		// INV Measures from Datalogger
		MesP 				: REAL ; 		(* (kW) 	Active Power output (AC) of inverter PCS01*)
		MesQ 				: REAL ;  		(* (kVAr)   Reactive AC Power Produced				  *)
		MesPdc 				: REAL ;  		(* (kW) 	Power measure (DC) of inverter			  *)
		MesIdc 				: REAL ;	 	(* (A) 	    Total Current measure (DC)				  *)
		MesUdc 				: REAL ;  		(* (V)  	Mean Voltage measure (DC)				  *)
		MesU 				: REAL ;		(* (V) 	    Mean Voltage measure (AC)				  *)
		MesV				: REAL ; 		(* (V)      Mean Phase to Neutral voltage			  *)
		MesI				: REAL ;		(* (A)      Mean Phase Current						  *)
		MesI0               : REAL ;        (* (A) 		Residual current						  *) 
		MesFreq				: REAL ; 		(* (Hz)     Frequency                                 *)
		MesS				: REAL ; 		(* (kVA)     Apparent Power						      *)
		MesInsuResistor		: REAL ; 		(* (kOhms) Insulation Resistance					  *)
		MesCosPhi			: REAL ; 		(* (p.u) Power Factor								  *)
		MesTemp				: REAL ; 		(* (C) Inverter Temperature							  *)
		MesState_Inv		: UINT ;		(* (NA) Inverter Status								  *)
		ParamPn				: REAL ; 		(* (kW) Nominal Capacity of SMA 25000 TL Inverter	  *)
		ParamQn				: REAL ;		(* (kVAr) Nominal reactive power 					  *)
		MesCurtl		    : BOOL ; 		(* (NA)Cal True if the inverter is curtailing Power	  *)
		MesAlarmCom			: BOOL ; 		(* (NA) Communication Alarm							  *)
		MesCP_Read			: BOOL := TRUE;	(* (NA) Cal : Permanent Condition for Read			  *)
		MesCP_Write			: BOOL := FALSE;	(* (NA) Cal : Permanenent Condition for Write		  *)
		                                                                                        
		MesOpened_Ac        : BOOL ;   		(* (NA) Ac switch is opened							  *)
		MesOpened_Dc        : BOOL ;   		(* (NA) Dc switch is opened							  *)
		                                                                                        
		OUT_CmdStart        : BOOL ;        (* (NA) OUT start command 							  *)
		OUT_CmdStop         : BOOL ;        (* (NA) OUT stop command   							  *)
		OUT_SetptPLimit    	: REAL ;        (* (kW) OUT P setpoint  							  *)
		OUT_SetptQ          : REAL ;        (* (kVAr)  OUT Q setpoint   						  *)
		MesState			: WORD ; 		(* (NA) Cal: Akuo Internal State . O=Stopped, 1 = RUN, 2 = Curtailment *)
		MesAlarmCode		: WORD ; 		(* (NA) Internal Akuo AlarmCode                       *)
		MesWarningCode		: WORD ; 		(* (NA) Internal Akuo WarningCode                     *)
		MesEventCode		: WORD ; 		(* (NA) Internal Akuo EventCode                       *)

END_STRUCT
END_TYPE

// ---- 01_Equipement_Library/Inverter/INV_DcModule.TcDUT
TYPE INV_DcModule :
STRUCT
	MesIdc				: REAL ; (* (A) Current of the Dc Module *)
	MesUdc				: REAL ; (* (V) Voltage of the Dc Module *)
	MesPdc				: REAL ; (* (kW) Power of the Dc Module *)
	MesClosed_DcSwitch	: BOOL ; (* (NA) Status of DC switch*)
	MesChargedSpring	: BOOL ; (* (NA) Status of string of DC switch*)
         		
	AX_STR				: ARRAY[1..CstNbSB_DcModule_G] OF STR;
END_STRUCT
END_TYPE

// ---- 01_Equipement_Library/Inverter/INV_DU.TcDUT
///////////
// Structure For Module. Main Operating Data to be saved (ex: OPC).  
//////////
TYPE INV_DU :
STRUCT
	
		MesI 				: REAL ; 		(* (dA) DU Current *)
		MesU 				: REAL ;  		(* (dV) DU Voltage *)
		MesIDState			: UINT ;		(* (NA) DU Status  *)
		
END_STRUCT
END_TYPE

// ---- 01_Equipement_Library/Inverter/INV_ABB_PVS.TcDUT
TYPE INV_ABB_PVS :
STRUCT
	MesData				: INV;		(* INV Object 									*)
	
	AX_STR				: ARRAY[1..12] OF STR;	(* STR Object 						*)
	
	MesI1				: REAL;		(* (A) Current Phase 1 							*)
	MesI2				: REAL;     (* (A) Current Phase 2 							*)
	MesI3				: REAL;     (* (A) Current Phase 3 							*)
	MesV1				: REAL;     (* (V) Voltage Phase 1 							*)
	MesV2				: REAL;     (* (V) Voltage Phase 2 							*)
	MesV3				: REAL;     (* (V) Voltage Phase 3 							*)
	MesU12				: REAL;     (* (V) Voltage between Phase 1 and 2 			*)
	MesU23				: REAL;     (* (V) Voltage between Phase 2 and 3 			*)
	MesU31				: REAL;     (* (V) Voltage between Phase 1 and 3 			*)
	MesPF				: REAL;     (* (NA) Power Factor							*)
	                                                                        		
	MesTemp_AC_cab		: REAL;		(* (C) Cabinet Temperature						*)
	MesTemp_HeatSink	: REAL;		(* (C) Heat Sink Temperature					*)
	MesState_InvWord	: WORD;		(* (NA)											*)
	MesVndOpeState		: UINT;		(* (NA) 										*)
	MesGlobalEvt		: WORD;		(* (NA) 										*)
	MesEacTot			: ULINT;	(* (NA) 										*)	
	MesEacDay			: LREAL;    (* (NA) 										*)
	
	MesEvent1 			: WORD;		(* (NA)											*)
	MesEventBitFld2 	: WORD;		(* (NA)											*)
	MesVndEventBitFld1 	: WORD;		(* (NA)											*)
	MesVndEventBitFld2 	: WORD;		(* (NA)											*)
	MesVndEventBitFld3 	: WORD;		(* (NA)											*)
	
	
	CmdP_Ack			: BOOL := TRUE;	(* (NA) P Command Acknowledge 				*)
	CmdQ_Ack			: BOOL := TRUE;	(* (NA) Q Command Acknowledge 				*)
	CmdPF_Ack			: BOOL;			(* (NA) Power Factor Command Acknowledge 	*)
	CmdStart_Ack		: BOOL := TRUE;	(* (NA) Start Command Acknowledge 			*)
	OUT_SetptCosPhi		: REAL := 1;	(* (NA) Power factor SetPoint Acknowledge	*)
	
END_STRUCT
END_TYPE

// ---- 01_Equipement_Library/Inverter/INV_Huawei.TcDUT
///////////
// Structure For Inverter. Main Operating Data to be saved ( ex: OPC ) .  
//////////
TYPE INV_Huawei :
STRUCT
	
	// INV Measures
		MesData				: INV ; (* INV *) 
                        	
		STR					: ARRAY[1..CstNbSB_INV_G ] OF STR ;  	(* STR *) 
		                	
		MesEDay				: REAL ;	    			(* (kWh)Daily Energy	*)
	    MesETot				: REAL ;					(* (kWh)Total Energy	*)
		MesI1				: REAL ;					(*	(A) MesI1			*)
		MesI2				: REAL ;					(*	(A) MesI2			*)
	    MesI3				: REAL ;					(*	(A) MesI3			*)
		MesU12				: REAL ;					(*	(V) MesU12			*)
        MesU23				: REAL ;					(*	(V) MesU23			*)
        MesU31				: REAL ;					(*	(V) MesU31			*)
		MesV1				: REAL ;					(*	(V) MesV1			*)
		MesV2				: REAL ;					(*	(V) MesV2			*)
		MesV3				: REAL ;					(*	(V) MesV3			*)
                        	                			
		MesStateIndic		: WORD ;					(*	(NA) Device status 		*)
		MesDeviceStatus		: WORD ;
// 0: standby , 1:grid connected , 2: grid connected normally , 3 : grid connection with derating due to power rationing , 4 grid connection with derating due to internal causes of the solar inverter
// 5 : normal stop , 6 : stop due to fault , 7 : stop due to power rationning , 8 : shutdown , 9 : spot check 


		MesOpeStatus 		: WORD ;					(*	(NA) MesOpeStatus 		*)
// 0 : locking status (0: locked; 1: unlocked) - 1 : PV Connection sttaus , 2 : DSP Data collection , 

		MesAlm1				: WORD ;					(*	(NA) MesAlm1				*)
		MesAlm2				: WORD ;					(*	(NA) MesAlm2				*)
		MesAlm3				: WORD ;					(*	(NA) MesAlm3				*)
	                                                        	
		MesID_DevStatus1	: WORD;						(* (NA) Akuo Created satus to compute device status alarms*)
		MesID_DevStatus2	: WORD;						(* (NA) Akuo Created satus to compute device status alarms*)
		


END_STRUCT
END_TYPE

// ---- 01_Equipement_Library/Inverter/INV_PE_HEMK.TcDUT
   ///////////
// Structure for PE Inverter. Main Operating Data to be saved (ex: OPC).  
//////////
TYPE INV_PE_HEMK:
STRUCT
	
	MesData					: INV ;				(* (NA) MesData*) 		            		
	// INV Measures
	AX_PowerCol				: ARRAY[1..CstNbPowerCol_INV_G ] OF PowerCol_INV_PE_HEMK; 			(* (NA) INV power columns *)
	AX_DcModule				: ARRAY[1..CstNbDcModule_INV_G] OF INV_DcModule; 			(* (NA) DC Inputs to the Inverter*)	
	
		
	//Electrical Measurements	
	MesAcDay				: UINT;				(* (kWh) Daily energy*)
	MesAcTot				: UINT;				(* (kWh) Total energy*)

	
	MesI1					: REAL; 			(* (A) Current phase 1 (R). INV: SV1.4 Grid current I1 (HEMK)															*)
	MesI2					: REAL; 			(* (A) Current phase 2 (S). INV: SV1.5 Grid current I2 (HEMK)															*)
	MesI3					: REAL; 			(* (A) Current phase 3 (T). INV: SV1.6 Grid current I3  (HEMK)															*)
	MesU12					: REAL; 			(* (V) Phase AB RMS voltage (line to line)at grid side of AC circuit breaker CB501. INV: SV1.1 Grid voltage RS (HEMK)	*)
	MesU23					: REAL; 			(* (V) Phase BC RMS voltage (line to line)at grid side of AC circuit breaker CB501. INV: SV1.2 Grid voltage ST(HEMK)	*)
	MesU31					: REAL; 			(* (V) Phase CA RMS voltage (line to line)at grid side of AC circuit breaker CB501. INV: SV1.3 Grid voltage TR (HEMK)	*)
	MesStatusCurtail_P		: WORD; 			(* (NA) P control : Cause of P control*)
	MesStatusCurtail_Q		: WORD; 			(* (NA) Q control : Cause of Q control*)
	MesDeratingGlobal		: REAL;				(* (%) Derating global taking into consideration IGBT Temp, Vdc et admission temp*)                               			
	                                			
	//Status Summary                			
	MesEventID				: REAL;				(* (NA) Event ID of the currently active event. 0= No event, 1 = Emergency stop, 3 = Remote emergency stop. SV8.15      *)
	MesIDFault				: UINT;				(* (NA) current fault ID check complete list in tab Failures*)	
	MesIDLastFaultedPowerCol: UINT;				(* (NA) Power Column ID of last alarm communicated*)	
	MesIDWarning			: UINT;				(* (NA) ID of current Warning : check complete list in tab Warnings*)	
	MesStateStart_Freq		: BOOL;				(* (NA) Start conditions Freq : True = Start OK*)
	MesStateStart_Vdc		: BOOL;				(* (NA) Start conditions Vdc : True = Start OK*)
	MesStateStart_MVCells	: BOOL;				(* (NA) Start conditions MVCells : True = Start OK*)
	MesStateStart_P			: BOOL;				(* (NA) Start conditions P : True = Start OK*)
	MesStateStart_Bbox		: BOOL;				(* (NA) Start conditions Bbox : True = Start OK*)
	
                            			
	MesSetptP				: REAL;				(* (%) Measurement of active power setpoint. INV: G8.1.3 P reference  	                                                *)                        	 
	MesSetptQ				: REAL;				(* (%) Measurement of reactive power setpoint. INV: G8.1.4 Q reference	                                   	            *)
	
	// System Commands
	ParamID_QMode			: UINT := 1; 		(* (NA) reactive power control mode : 0: Cos Phi, 1: Q,  2: I, 4: V/Q mode   G8.1.2 register: 40551  		*)
	ParamID_PMode			: UINT := 1; 		(* (NA) active power control mode : 0: MPPt, 1: I, 2: P, 3: Vdc										 		*)
		                                    	                                                                                                         		
	MesCP_Start        		: BOOL;				(* (NA) Start conditions. INV: SV4.3.1-Start conditions all											 		*)                 		        		
	                                                                                                         											
	// Inverter's Control Cabinet  Status                                                                       											
	MesTemp_Internal		: REAL; 		 	(* (C) Control cabinet temperature. INV: SV4.1.4 Internal temperature										*)
	MesTemp_Control			: REAL; 		 	(* (C) Control cabinet temperature. INV: SV4.1.4 Internal temperature										*)
	MesTemp_IGBTmax			: REAL; 		 	(* (C) Maximum IGBT temperature. INV: SV4.1.5 Max IGBTs temperature											*)
	MesTemp_PowerColmax		: REAL; 		 	(* (C) Maximum power column temperature. INV: SV4.1.6 Max modules temperature								*)
	MesAlarm_Control		: UINT;			 	(* (NA) Control cabinet alarm. INV: SV4.1.1 Current fault 													*) 
	MesWarning_Control		: UINT;			 	(* (NA) Control cabinet warning. INV: SV4.1.2 Current warning					    						*)			
	MesState_Control 		: UINT;			 	(* (NA) Control cabinet state. INV: SV4.1.3 Current status													*)
	MesState_Module			: WORD;				(* (NA) Status of modules*)	 
	MesNbRunningModules		: UINT;				(* (NA) Number of running modules*)
                                        	                                                    	                                						
	// Reset command                         	                                                    	                                						
	OUT_CmdReset 			: BOOL; 		 	(* (NA) OUT reset command. INV: Reset command 43012															*)

	MesP_LV					: REAL;				(* (kW) LV Active Power*)
	MesQ_LV					: REAL;				(* (kVAr) LV Reactive Power*)
	MesS_LV					: REAL;				(* (kVA) LV Apparent Power*)
	MesCosPhi_LV			: REAL;				(* (NA) LV CosPhi*)
    MesU12_LV				: REAL; 			(* (kV) LV Voltage 12*)                                                                              															
    MesU23_LV				: REAL; 			(* (kV) LV Voltage 23*)                                                                              															
    MesU31_LV				: REAL; 			(* (kV) LV Voltage 31*)                                                                              															
	MesI1_LV				: REAL; 			(* (A) Current phase 1 (R). INV: SV1.4 Grid current I1 (HEMK)															*)
	MesI2_LV				: REAL; 			(* (A) Current phase 2 (S). INV: SV1.5 Grid current I2 (HEMK)															*)
	MesI3_LV				: REAL; 			(* (A) Current phase 3 (T). INV: SV1.6 Grid current I3  (HEMK)															*)
	MesPAvailable			: REAL;
	MesPn					: REAL;

	
	MesEventCode2			: WORD ; 


END_STRUCT
END_TYPE

// ---- 01_Equipement_Library/Inverter/INV_PE_HEMG3.TcDUT
///////////
// Structure for PE Inverter. Main Operating Data to be saved (ex: OPC).  
//////////
TYPE INV_PE_HEMG3:
STRUCT
	
	// INV Measures
	MesData					: INV ;	(* (NA) MesData 																										*) 		            		
	// Power column (PE name : Modules) 
	AX_PowerCol				: ARRAY[1..6] OF PowerCol_INV_PE_HEMG3;	(* (NA) Power column of the PE Skid  *) 
	AX_DU 					: ARRAY[1..CstNb_DU_G] OF INV_DU; (* (NA) Disconnecting Units Channels *)
	
	//Electrical Measurements	
	MesI1					: REAL; (* (A) Current phase 1 (R). INV: SV1.4 Grid current I1 (HEMK)															*)
	MesI2					: REAL; (* (A) Current phase 2 (S). INV: SV1.5 Grid current I2 (HEMK)															*)
	MesI3					: REAL; (* (A) Current phase 3 (T). INV: SV1.6 Grid current I3  (HEMK)															*)
	MesU12					: REAL; (* (V) Phase AB RMS voltage (line to line)at grid side of AC circuit breaker CB501. INV: SV1.1 Grid voltage RS (HEMK)	*)
	MesU23					: REAL; (* (V) Phase BC RMS voltage (line to line)at grid side of AC circuit breaker CB501. INV: SV1.2 Grid voltage ST(HEMK)	*)
	MesU31					: REAL; (* (V) Phase CA RMS voltage (line to line)at grid side of AC circuit breaker CB501. INV: SV1.3 Grid voltage TR (HEMK)	*)
	MesPconnected			: REAL; (* (%) Current available active power. INV: SV4.2.1 P limit inst 														*)                                                     									
	MesStatusCurtail_P		: WORD; 			(* (NA) P control : Cause of P control*)
	MesStatusCurtail_Q		: WORD; 			(* (NA) Q control : Cause of Q control*)
	MesInsuResistor_AC		: REAL;	(* (Ohms) AC Insulation Resistance. INV: SV3.2.2  Resistor 																*)
	OUT_CmdInvLocal			: BOOL; (*determine whether setpoint is from local or remote *)
	
	
	
	//Communication Status                                                                                              									
	MesStateCom				: BOOL; (* (NA) Cal: False := Not communicating, True := Communicating	 														*)
	
	//Status Summary
	MesStateCBac			: BOOL; (* (NA) False := Open, True := Close, Status of event139 "CB501 Closed". AC circuit breaker CB501 is closed 			*)
	MesStateCBdc			: BOOL; (* (NA) False := Open, True := Close, Status of event140 "CB201 Closed". DC circuit breaker CB201 is closed             *)
	MesEarthing_Relay		: BOOL; (* (NA) False := Open, True := Close, Status of event157 "K202 Closed". Ground relay K202 is closed                     *)
	MesFaultGnd				: BOOL; (* (NA) False := Alert, True := No alert, Ground fault status. Digital outputDO_121 follows the state of this register  *)
	MesStateNoAlert			: BOOL; (* (NA) False := Alert iverter has detected an abnormal event which prevents operation. ; True := No alert.             *)
	MesState				: UINT; (* (NA) This parameter should be used for informational status only                                                     *)
	MesAlarmID				: UINT; (* (NA) Fallo actual *)
	MesWarningID			: UINT; (* (NA) Warning actual*)


	MesBdrigeCtlMod			: UINT;	(* (NA) Inverter bridge control mode                                                                                    *)
	MesWorkingHr			: REAL; (* (Hr) Total duration that the inverter has been online since power up                                                 *)
	MesEventID				: REAL;	(* (NA) Event ID of the currently active event. 0= No event, 1 = Emergency stop, 3 = Remote emergency stop. SV8.15      *)
	
	MesSetptP				: REAL;	(* (%) Measurement of active power setpoint. INV: G8.1.3 P reference  	                                                *)                        	 
	MesSetptQ				: REAL;	(* (%) Measurement of reactive power setpoint. INV: G8.1.4 Q reference	                                   	            *)
	MesSetptCosPhi			: REAL; (* (pu) Measurement of power factor setpoint. INV: G8.1.4 Cos phi reference                                	            *)
	MesStartDisabled		: BOOL; (* (NA) Start disable : False := Start can be abled 						 											*)
	
	// System Commands
	ParamID_QMode			: UINT := 1; 		(* (NA) reactive power control mode : 0: Cos Phi, 1: Q,  2: I, 4: V/Q mode   G8.1.2 register: 40551  		*)
	ParamID_PMode			: UINT := 1; 		(* (NA) active power control mode : 0: MPPt, 1: I, 2: P, 3: Vdc										 		*)
		                                    	                                                                                                         		
	MesCP_Start        		: BOOL;				(* (NA) Start conditions. INV: SV4.3.1-Start conditions all											 		*)                 		        		
	                                                                                                         											
	// Inverter's Control Cabinet  Status                                                                       											
	MesTemp_DU				: REAL;			 	(* (C) Disconnecting unit temperature. INV: SV4.1.4b DU Internal  											*)
	MesTemp_Control			: REAL; 		 	(* (C) Control cabinet temperature. INV: SV4.1.4 Internal temperature										*)
	MesTemp_IGBTmax			: REAL; 		 	(* (C) Maximum IGBT temperature. INV: SV4.1.5 Max IGBTs temperature											*)
	MesTemp_PowerColmax		: REAL; 		 	(* (C) Maximum power column temperature. INV: SV4.1.6 Max modules temperature								*)
	MesAlarm_Control		: UINT;			 	(* (NA) Control cabinet alarm. INV: SV4.1.1 Current fault 													*) 
	MesWarning_Control		: UINT;			 	(* (NA) Control cabinet warning. INV: SV4.1.2 Current warning					    						*)			
	MesState_Control 		: UINT;			 	(* (NA) Control cabinet state. INV: SV4.1.3 Current status													*)
	                                         	                                                    	                                						
	// Reset command                         	                                                    	                                						
	OUT_CmdReset 			: BOOL; 		 	(* (NA) OUT reset command. INV: Reset command 43012															*)
	OUT_CmdEmergencyStop	: BOOL; 		 	(* (NA) OUT emergency stop command. INV: Emergengy stop command 43200										*) 
	MesNbRunningModules		: REAL; 			(* (NA) Number of modules running*)

    MesEventCode2			: WORD ;                                                                                     															
END_STRUCT
END_TYPE

// ---- 01_Equipement_Library/Inverter/SKID_PE_HEMG3.TcDUT
///////////
// Structure for PE SKID. Main Operating Data to be saved (ex: OPC).  
//////////
TYPE SKID_PE_HEMG3:
STRUCT
	
	MesCP_Read							: BOOL := TRUE;		(* (NA) Cal : Permanent Condition for Read		*)
	MesCP_Write							: BOOL := TRUE;		(* (NA) Cal : Permanenent Condition for Write   *)
	
	MesDisparoTemp_Transformador1 		: BOOL; (* (NA) alarm transformer*)
	MesAlarmTemp_Transformador1	 		: BOOL; (* (NA) warning temp transformer*)
	MesDisparoPresion_Transformador1 	: BOOL; (* (NA) alarm pressure transformer*)
	MesDisparoOil_Transformador1 		: BOOL; (* (NA) alarm oil transformer*)

	MesDisparoTemp_Transformador2 		: BOOL; (* (NA) alarm transformer*)
	MesAlarmTemp_Transformador2	 		: BOOL; (* (NA) warning temp transformer*)
	MesDisparoPresion_Transformador2 	: BOOL; (* (NA) alarm pressure transformer*)
	MesDisparoOil_Transformador2 		: BOOL; (* (NA) alarm oil transformer*)

	MesSeccionador1_Abierto				: BOOL; (* (NA) Secc opened*)
	MesEarth1_Abierto					: BOOL; (* (NA) Earth switch Opened opened*)
	MesMonitorGas						: BOOL; (* (NA) *)
	MesMonitorGas2						: BOOL; (* (NA) *)
	MesSeccionador2_Abierto				: BOOL; (* (NA) Secc opened*)
	MesEarth2_Abierto					: BOOL; (* (NA) Earth switch Opened opened*)
	MesSeccionadorMain1_Abierto			: BOOL; (* (NA) Secc opened*)
	MesEarthMain1_Abierto				: BOOL; (* (NA) Earth switch Opened opened*)
	MesCb1_Abierto						: BOOL; (* (NA) Circuit breaker*)
	MesProtectRelay1_fallo				: BOOL; (* (NA) protect relay fault*)
	MesProtectRelay1_overvoltage		: BOOL; (* (NA) protect relay fault*)
	MesProtectRelay1_springloaded		: BOOL; (* (NA) *)

	MesSeccionadorMain2_Abierto			: BOOL; (* (NA) Secc opened*)
	MesEarthMain2_Abierto				: BOOL; (* (NA) Earth switch Opened opened*)
	MesCb2_Abierto						: BOOL; (* (NA) Circuit breaker*)
	MesProtectRelay2_fallo				: BOOL; (* (NA) protect relay fault*)
	MesProtectRelay2_overvoltage		: BOOL; (* (NA) protect relay fault*)
	MesProtectRelay2_springloaded		: BOOL; (* (NA) *)

	MesTemp1							: REAL;(* (°C) temperature of the transformer*)
	MesTemp2							: REAL;(* (°C) temperature of the transformer*)
	
	MesAlarmCom							: BOOL;
	MesAlarmCode						: WORD; 			(* (NA) Internal Akuo AlarmCode                 *)
	MesWarningCode						: WORD; 			(* (NA) Internal Akuo WarningCode               *)
	MesEventCode						: WORD;		 		(* (NA) Internal Akuo EventCode                 *)                                                                            															
END_STRUCT
END_TYPE

// ---- 01_Equipement_Library/Inverter/PowerCol_INV_PE_HEMK.TcDUT
///////////
// Structure For Module. Main Operating Data to be saved (ex: OPC).  
//////////
TYPE PowerCol_INV_PE_HEMK :
STRUCT
		MesData				: PowerCol_INV ; 	
		
		
		MesS 				: REAL ;  		(* (kVA)   Apparent power output of the power column 													*)
		MesU12				: REAL ;		(* (A) 		Module Voltage																				*)
		MesU23				: REAL ;		(* (A) 		Module Voltage																				*)
		MesU31				: REAL ;		(* (A) 		Module Voltage																				*)
		
		ParamUn				: REAL ;		(* (V) 		Nominal AC voltage (SV4.4.4.1.2)																		*)
		ParamImax			: REAL ; 		(* (A) 		Nominal AC current (SV4.4.4.1.7)																		*) 
		ParamVdcn			: REAL ;        (* (V) 		Nominal DC voltage (SV4.4.4.1.6)																		*)
		ParamIdcmax			: REAL ;        (* (A) 		Nominal DC current (SV4.4.4.1.8)																		*)
		ParamSn				: REAL ;        (* (kVA) 	Nominal apparent power (SV4.4.4.1.3)																	*)
		
		MesTemp				: REAL ;		(* (C) 		Ambient temperature of the selected module																*)
		MesTempmax			: REAL ;		(* (C) 		Maximum IGBT temperature of the selected module															*)
		MesHygro			: REAL ; 		(* (%) 		Percentage of humidity																					*)
		
		MesStateIO			: WORD ;		(* (NA) 	0: Open, 1: Closed. Bit 1 =  fan contactor, Bit 2 = main AC contactor, Bit 3 = AC soft charge contactor, Bit 4 = LCL filter contactor, Bit 5 = DC contactor , Bit 6 = reserved, Bit 7 = if open : overheating in the coil, Bit 8 = fan contactor feedback, Bit 9 = AC main contactor feedback, Bit 10 = AC soft charge contactor feedback, Bit 11 = LCL filter contactor feedback , Bit 12 = DC contactor feedback *) 		
		MesState			: UINT ;		(* (NA) 	Module status (SV9.3 PE documentation p.97)																*)
		
		MesEActProd			: REAL ;		(* (kWh) 	Total amount of  generated energy since commissioning 													*)
		MesEReactProd		: REAL ;		(* (kVarh)  The amount of reactive energy generated since commissioning 											*) 	   
	
END_STRUCT
END_TYPE

// ---- 01_Equipement_Library/Inverter/PowerCol_INV_PE_HEMG3.TcDUT
///////////
// Structure For Module. Main Operating Data to be saved (ex: OPC).  
//////////
TYPE PowerCol_INV_PE_HEMG3 :
STRUCT
		MesData				: PowerCol_INV ; 	

													
		
		ParamUn				: REAL ;		(* (V) 		Nominal AC voltage (SV4.4.4.1.2)																		*)
		ParamImax			: REAL ; 		(* (A) 		Nominal AC current (SV4.4.4.1.7)																		*) 
		ParamVdcn			: REAL ;        (* (V) 		Nominal DC voltage (SV4.4.4.1.6)																		*)
		ParamIdcmax			: REAL ;        (* (A) 		Nominal DC current (SV4.4.4.1.8)																		*)
		ParamSn				: REAL ;        (* (kVA) 	Nominal apparent power (SV4.4.4.1.3)																	*)
		
		MesTemp				: REAL ;		(* (C) 		Ambient temperature of the selected module																*)
		MesTempmax			: REAL ;		(* (C) 		Maximum IGBT temperature of the selected module															*)
		MesHygro			: REAL ; 		(* (%) 		Percentage of humidity																					*)
		
		MesStateIO			: WORD ;		(* (NA) 	0: Open, 1: Closed. Bit 1 =  fan contactor, Bit 2 = main AC contactor, Bit 3 = AC soft charge contactor, Bit 4 = LCL filter contactor, Bit 5 = DC contactor , Bit 6 = reserved, Bit 7 = if open : overheating in the coil, Bit 8 = fan contactor feedback, Bit 9 = AC main contactor feedback, Bit 10 = AC soft charge contactor feedback, Bit 11 = LCL filter contactor feedback , Bit 12 = DC contactor feedback *) 		
		MesState_Inv		: UINT ;		(* (NA) 	Module status (SV9.3 PE documentation p.97)																*)
		MesState_Inv_ID		: WORD;			(* (NA)		Calculated tag to create alarms for the State_Inv*)
		MesState_Inv_ID2	: WORD;			(* (NA)		Calculated tag to create alarms for the State_Inv*)
		MesEActProd			: REAL ;		(* (kWh) 	Total amount of  generated energy since commissioning 													*)
		MesEReactProd		: REAL ;		(* (kVarh)  The amount of reactive energy generated since commissioning 											*) 	   
	                 															

END_STRUCT
END_TYPE

// ---- 01_Equipement_Library/Inverter/INV_SmaSCXXXCP_HE.TcDUT
TYPE INV_SmaSCXXXCP_HE :
	//SMA CP, CP-US, CP-JP and HE-20
STRUCT
		Mesdata					: INV;
		BJMonitor					: ARRAY[1..CstNbSB_INV_G] OF JuncBox;	

// Device Family
		MesEventID				: REAL;		(* Event ID of the current event [ErrNo]*)
		MesWaitGridTm			: TIME; 	(* Time until grid connection attempt (s) [TmsRmg].*)
	// Setpoint ??? RecoAction
		SetptRecoAction			: REAL;		(* 336 = Contact the manufacturer,337 = Contact the installer,338 = Invalid [Prio]*)
		MesOpened_CBGrid		: BOOL;     (* 51 = Contactor closed,311 = Contactor open [GriSwStt]*)
		MesRiso					: REAL;		(* Insulation resistance (Ohm) [Riso]*)
		MesState_KeyComut		: BOOL;     (* Status of key switch :381 = Stop,569 = Activated [DInKeySwStrStp]*)
		MesState_Inv			: REAL;		(* Operating state, 309 = Operation,381 = Stop,455 = Warning,1392 = Error,1393 = Wait for PV voltage,1394 = Wait for AC grid,1480 = "Wait for electricity supplier" operating state (for 0% regulation),1560 = Remote shutdown active,2383 = Manual restart [mode]*)
		MesIDError				: REAL;     (* Error location OF the present error,267 = Inverter , 1395 = DC section,1396 = AC grid [Error]*)
		MesEventID_INVSMA		: REAL;		(* Current, complete event number [ErrNoSma]*)
		MesOpened_GFDI			: BOOL;     (* Switching status of the GFDI  (311: Open & 51 : Close) [DInGfdi]*)
		MesOpened_CBdc			: BOOL;		(* DC Switch status (51: Close, 311: Open) [DcSwStt]*)
		MesState_Restart		: REAL;		(* Status of current restart interlock :1690 = Fast shut-down, 2386 = Overvoltage, 2387 = Undervoltage, 2388 = Overfrequency, 2389 = Underfrequency, 2390 = Passive islanding detection, 2490 = Phase lost detection [ManResStt]*)
		MesOpened_CBac			: BOOL;  	(* AC switch-disconnector in cabinet [AcDiscon]: 51 = Closed, 311 = Open*)
		MesEActTot				: REAL;     (* Total yield (MWh) [E-Total]*)
		MesEActDay				: REAL;     (* Daily yield (Wh) [E-heute]*)
		MesWorkingHr			: TIME;     (* Operating time (Hr) [h-On]*)
		MesFeedTm				: TIME;     (* Feed-in Time (Hr) []*)
		MesWorkingHr_Fan1		: TIME;     (* Operating time of the interior fan 1 (Hr) [CntFanCab1]*)
		MesWorkingHr_Fan2		: TIME;     (* Operating time of the interior fan 2 (Hr) [CntFanCab2]*)
		MesWorkingHr_Heat		: TIME;		(* Operating time of the interior heater (Hr) [CntFanHs]*)
		MesWorkingHr_Heat2		: TIME;		(* Operating time of the interior heater (Hr) [CntHtCab2]*)
		MesWorkingHr_Fan3		: TIME;     (* Operating time of interior fan 3 (h) [CntFanCab3]*)
		MesU12					: REAL;     (* (V) Line to line Voltage L1-L2 utility grid VacL12*)
		MesU23					: REAL;     (* (V) Line to line Voltage L2-L3 utility grid VacL23*)
		MesU31					: REAL;     (* (V) Line to line Voltage L3-L1 utility grid VacL31*)
		MesI1					: REAL;		(* (A) Mean AC current L1 Total [IacL1]*)
		MesI2					: REAL;		(* (A) Mean AC current L2 Total [IacL2]*)
		MesI3					: REAL;		(* (A) Mean AC current L3 Total [IacL3]*)
		MesTypeCosPhi			: REAL;		(* Setpoint excitation type of cos φ [PF-PFExtSpt]: 1041 = Capacative, 1042 = Inductive*)
		MesQMode	           	: REAL;		(* Operating mode of the reactive power regulation [Q-VArMod]:303 = Off,1069= Reactive power-/voltage characteristic curve Q(V),1070 = Reactive power Q, direct setpoint,1071 = Reactive power const. Q (kVAr)                                                          *)
											(* 1072 = Reactive power Q, setpoint via system control, 1074 = cos φ, direct setpoint, 1075 = cos φ, setpoint via system control, 1076 = cos φ(P) – characteristic curve, 1387 = Reactive power Q, setpoint via analog input , 1388 =cos φ, setpoint via analog input, *)
											(* 1389 = Reactive power-/voltage characteristic curve Q(V) with hysteresis and deadband*)
		MesSetptQ				: REAL;     (* Reactive power setpoint (kVAr) [SpntPwrRt]*)
		MesSetptQ_Pct			: REAL;     (* Reactive power setpoint (%) [Q-VArNom].*)
		MesSetptCosPhi			: REAL;		(* Setpoint cos φ [PF-PFSpt]*)
		MesSetptType_CosPhi		: REAL;		(* Setpoint excitation type of cos φ [PF-PFExtSpt]: 1041 = Capacative, 1042 = Inductive*)
		MesPMode				: REAL;		(*	 [P-WMod]: 303 = Off, 1077 = Active power limitation P (kW), 1078 = Active power limitation P in (%) of PMAX,*)
											(*	1079 = Active power limitation P via plant control, 1390 = Active power limitation P via analog input*)

// Stopped here											(*	1391 = Active power limitation P via digital inputs*)
		MesPSetpt				: REAL;     (* (kW) Active power setpoint [P-WSp]*)
		MesPSetptPct			: REAL;     (* (%) Active power setpoint  [P-WNom].*)
		MesTmpHs				: REAL;		(* (°C) Heat sink temperature 1 [TmpHs]*)
		MesTmpCab1				: REAL;		(* (°C) Heat sink temperature Cab 1 [TmpCab1]*)
		MesTmpCab3				: REAL;		(* (°C) Heat sink temperature Cab 3 [TmpCab3]*)
		MesTmpExt				: REAL;		(* (°C) External temperature 1 [TmpExt1]*)
		MesTmpCol				: REAL;		(* (°C) Temperautre of the sinusoidal filter choke [TmpCol]*)
		MesGHI					: REAL;		(* (W/m²) Total irradiation of the sensor surface [ExtSolIrr]*)
		MesInCur1				: REAL;		(* (mA) Analog current Input 1 [ExtSolIrr]*)
		MesInCur2				: REAL;		(* (mA) Analog current Input 2 [ExLAnaInCur]*)
		MesOpStateOn			: BOOL;		(* (NA) Operating state : 381 = Stop,569 = Activated  [SpntRemEna]*)
		MesbRIsoOn				: BOOL;		(* (NA) External measurement of the insulation resistance : 303=Off, 308=On*)
		//AX_BJ					: ARRAY [1..8] OF REAL; // (A) Current of each BJ*)

END_STRUCT
END_TYPE

// ---- 01_Equipement_Library/Inverter/INV_ClusterPowerOne.TcDUT
///////////
// Structure For Inverter. Main Operating Data to be saved ( ex: OPC ) .  
//////////
TYPE INV_ClusterPowerOne :
STRUCT
		MesAlarmCode		: WORD ; 		(* (NA) Internal Akuo AlarmCode                       *)
		MesWarningCode		: WORD ; 		(* (NA) Internal Akuo WarningCode                     *)
		MesEventCode		: WORD ; 		(* (NA) Internal Akuo EventCode                       *)


		MesAlarmCom			: BOOL ; 		(* (NA) Communication Alarm							  *)
	
		AX_INV : ARRAY [1..3] OF INV_PowerOne ; (*  INV Object *)

		MesNbInvConnected 					: UINT ; (* Cal Number of inverters connected *)
		MesState						: UINT ;		(* (NA) Akuo Standardized 								  *)
		
		OUT_CmdStart        : BOOL ;        (* (NA) OUT start command 							  *)
		OUT_CmdStop         : BOOL ;        (* (NA) OUT stop command   							  *)
		OUT_SetptP    	    : REAL ;        (* (kW) OUT P setpoint  							  *)
		OUT_SetptTanPhi         : REAL ;    (* (p.u)  OUT TanPhi setpoint   					   *)
		
		
		
		
		
END_STRUCT
END_TYPE

// ---- 01_Equipement_Library/Inverter/INV_Jema_IFX6.TcDUT
TYPE INV_Jema_IFX6 :
STRUCT
		MesData					: INV; (* Child Structure*)

		AX_PowerCol				: ARRAY[1..3] OF PowerCol_INV_Jema;(* Child Structure*)
		AX_STR					: ARRAY[1..24] OF STR;(* Child Structure*)
		
		MesEacTot				: REAL;     (* (kWh)Total yield [E-Total]*)
		MesEacDay				: REAL;     (* (kWh)Daily yield [E-heute] *)
                            	
		MesGFDI					: WORD; 	(* (NA) GFDI reset:after set1 to reset set0 again *)		
		                    	
		MesI1					: REAL;		(* (A) Current in phase 1*)
		MesI2 					: REAL;     (* (A) Current in phase 2*)
		MesI3					: REAL;     (* (A) Current in phase 3*)
		                    	
		MesTmpPlant				: REAL;		(* (°C) temperature in Plant*)
		MesTmpExt1				: REAL;     (* (°C) External temperature 1 *)
		MesTmpExt2				: REAL;     (* (°C) External temperature 2 *)
		MesTmp					: REAL;     (* (°C) Temperature *)
		MesTmpPlc				: REAL;     (* (°C) Temperature of PLC*)
		MesHygroPlc				: REAL;     (* (%) Hygrometry of PLC*)
		
		                    	
		MesVdc1					: REAL;		(* (V) Voltage of DC entry*)
		MesVdc2					: REAL;     (* (V) Voltage of DC entry*)
		MesVdc3					: REAL;     (* (V) Voltage of DC entry*)
		                    	
		MesPLC_IN1				: WORD;		(* (NA) PLC inputs *)
		MesPLC_IN2				: WORD;     (* (NA) PLC inputs *)
		                    	
		MesPowerColConnected_ALO : BOOL;		(* (NA) At least one power column connected*)	
		MesNbPowerCol_Connected	: UINT ; (* (NA) Number of power column connected*)	
		OUT_CmdHeartBeat		: BOOL;			(* (NA) Heartbit*)
		OUT_CmdP				: BOOL := TRUE;		(* (NA) Command to activate P regulation*)
		OUT_CmdQ				: BOOL := TRUE;     (* (NA) Command to activate Q regulation*)
		OUT_CmdPF				: BOOL;             (* (NA) Command to activate PF regulation*)
		OUT_CmdStart			: BOOL := TRUE; 	(* (NA) Start order (1: Start)*)
		OUT_CmdCells			: BOOL;				(* (NA) Close Cells (1: Close)*)
		OUT_CmdPvF				: BOOL;				(* (NA) Command to active PvF regulation*)	
		OUT_CmdQvU				: BOOL;             (* (NA) Command to active QvU regulation*)	
		OUT_CmdResetGFDI		: BOOL;				(* (NA) Command to reset GFDI*)
		                    	
		OUT_CmdControl			: WORD;			 	(* (NA) Control word to send to the INV*)
			                	                    
		OUT_SetptP				: REAL;             (* (kW) P Setpoint sent to the inverters*)
		OUT_SetptQ				: REAL;             (* (kW) Q Setpoint sent to the inverters*)
		OUT_SetptQMax			: REAL;				(* (kW) Max Q setpoint*)
        OUT_SetptQMin       	: REAL;        	    (* (kW) Min Q setpoint*)
		OUT_SetptPF				: REAL;			    (* (kW) PF Setpoint sent to the inverters *)
			                                        
		
END_STRUCT
END_TYPE

// ---- 01_Equipement_Library/Inverter/INV_PowerOne.TcDUT
///////////
// Structure For Inverter. Main Operating Data to be saved ( ex: OPC ) .  
//////////
TYPE INV_PowerOne :
STRUCT
		MesData				: INV ; (* MesData *)
	

	// INV Measures
		MesEDay				: REAL;     (* (kWh)	Daily Energy*)
	    MesETot				: REAL;		(* (kWh)    Total Energy*)
	    MesEPartial			: REAL;		(* (kWh)	??? To check*)
	    MesEWeek			: REAL;		(* (kWh)	Week Energy*)
	    MesEMonth			: REAL;		(* (kWh)	Monthly Energy*)
	    MesEYear			: REAL;     (* (kWh)	Yearly Energy*)
			
		MesNbPowerColConnected				: UINT ; (* Cal Number of powercolumns connected *)
	//Modules Measures
		AX_PowerCol 	: ARRAY[1..6] OF PowerCol_INV_Power_One; 	(* PowerCol Object  *)
	

END_STRUCT
END_TYPE

// ---- 01_Equipement_Library/Inverter/INV_Sch4400.TcDUT
///////////
// Structure For Inverter. Main Operating Data to be saved (ex: OPC).  
//////////
TYPE INV_Sch4400 :
STRUCT
	
	// INV Measures
	MesData					: INV ;					(* MesData *) 
		            		
	AX_STR						: ARRAY[1..10] OF STR;	(* (NA) Strings *)

	//Electrical Measurements
	MesI1					: REAL; (* (A) Phase A RMS current at inverter side of AC circuit breaker CB501								*)
	MesI2					: REAL; (* (A) Phase B RMS current at inverter side of AC circuit breaker CB501                             *)
	MesI3					: REAL; (* (A) Phase C RMS current at inverter side of AC circuit breaker CB501                             *)
	MesV1					: REAL; (* (V) Phase A RMSvoltage (line to virtual neutral)at grid side of AC circuit breaker CB501         *)
	MesV2					: REAL; (* (V) Phase B RMSvoltage (line to virtual neutral)at grid side of AC circuit breaker CB501         *)
	MesV3					: REAL; (* (V) Phase C RMSvoltage (line to virtual neutral)at grid side of AC circuit breaker CB501         *)
	MesU12					: REAL; (* (V) Phase AB RMS voltage (line to line)at grid side of AC circuit breaker CB501                  *)
	MesU23					: REAL; (* (V) Phase BC RMS voltage (line to line)at grid side of AC circuit breaker CB501                  *)
	MesU31					: REAL; (* (V) Phase CA RMS voltage (line to line)at grid side of AC circuit breaker CB501                  *)
	
	//Production Measurements
	MesEActProd				: REAL; (* (Wh) Active energy delivered.Integrates positive values of GenMMTR/DmdWhFil.Ignores negative values		*)
	MesEActCons				: REAL; (* (Wh) Active energy consumed.Integrates negative values of GenMMTR/DmdWhFil.Ignores positive values       *)
	MesEReactProd			: REAL; (* (VArh) Reactive energy delivered.Integrates positive values of GenMMTR/DmdVAhFil.Ignores negative values *)
	MesEReactCons			: REAL; (* (VArh) Reactive energy consumed.Integratesnegative values of GenMMTR/DmdVAhFil.Ignores positive values   *)
	MesEday					: REAL; (* (Wh) Active energy produced during the day                                                               *)
	
	//Communication Status
	MesStateCom				: BOOL; (* (NA) False := Not communicating, True := Communicating 	*)
	
	//Status Summary
	MesStateCBac			: BOOL; (* (NA) False := Open; True := Close, Status of event139 "CB501 Closed". AC circuit breaker CB501 is closed /INVx/AcXCBR/ClsActVal				 *)
	MesStateCBdc			: BOOL; (* (NA) False := Open; True := Close, Status of event140 "CB201 Closed". DC circuit breaker CB201 is closed /INVx/DcXCBR/ClsActVal               *)
	MesEarthing_Relay		: BOOL; (* (NA) False := Open; True := Close, Status of event157 "K202 Closed". Ground relay K202 is closed /INVx/GndXSWI/ClsActVal                      *)
	MesFaultGnd				: BOOL; (* (NA) False := Alert; True := No alert, Ground fault status. Digital outputDO_121 follows the state of this register /INVx/RcdMMXU/GndFltDrvSt *)
	MesStateNoAlert			: BOOL; (* (NA) False := Alert iverter has detected an abnormal event which prevents operation. ; True := No alert. /INVx/GenGGIO/NoFltDrvSt             *)
	MesState				: UINT; (* (NA) This parameter should be used for informational status only //INVx/GenZINV/Stt                                                           *)
	MesBdrigeCtlMod			: UINT;	(* (NA) Inverter bridge control mode /INVx/GenZINV/CtlMod                                                                                        *)
	MesWorkingHr			: REAL; (* (Hr) Total duration that the inverter has been online since power up /INVx/GenGAPC/TmsCnt                                                	 *)
	MesEvendID				: REAL;	(* (NA) Event ID of the currently active event. /INVx/EvtGGIO/ActId                                                                              *)
	MesEventID_Stop			: REAL;	(* (NA) Event ID of the first event that caused the Inv to go offline (normal or not)/INVx/EvtGGIO/OflStrActId                                   *)
	MesStateID_Recovery		: REAL;	(* (NA) Procedure for the Inv to recover: 0:No stop event, 1:Automatic, 2:Manual (=acknowledge), 3:Local (= physique) /INVx/EvtGGIO/RecovActTyp  *)
	MesEventID_AbnormalOff	: REAL;	(* (NA) Abnormal offline status ID: ID of the event that caused an abnormal stop (0=No abnormal stop) /INVx/EvtGGIO/OflForcSt                    *)
	MesState_TypeSetptP		: REAL;	(* (NA) Dominant limit or setpoint affecting active power production : 0: None, 11: CmdSetpt from comm, 15: MPPT /INVx/WMMXU/PriConId            *)
	MesSetptP				: REAL;	(* (pu) Value of the dominant active power limit W                                                                                    			 *)
	MesState_TypeSetptQ		: REAL; (* (NA) Dominant limit or setpoint affecting reactive power production : 0: None, 6: CmdSetpt from comm                                     	 *)
	MesSetptQ				: REAL;	(* (pu) Value of the dominant reactive power limit VAr                                                                                			 *)
	
	MesStartDisabled		: BOOL; (* (NA) Start disable : False := Start can be abled 						 *)
	MesStartDisabledPersis	: BOOL; (* (NA) Persistent start disable : must be the same as MesStartDisabled      *)
	
	// System Commands
	// Persistent value of inverter enable command.The value set here defines the initial value of GenZINV/Ena when the inverter powers on
	MesSetptP_CC 			: REAL;			(* (kW)   value of active power COMMAND																 *)
	MesSetptQ_CC 			: REAL;			(* (kVar) value of reactive power COMMAND                                                            *)
	MesSetptCosPhi_CC 		: REAL; 		(* (NA)  Power factor                                                            					 *)
	ParamID_QType			: UINT := 1; 	(* (NA) reactive power is defined by : 1: Q command mode, 2: PF command mode, 3: Q(P) command mode   *)
	ParamTP_RampP			: REAL; 		(* (s) Duration for the active power to reach the new setpoint                 						 *)
	ParamTP_RampCosPhi		: REAL; 		(* (s) Duration for the active power to reach the new setpoint                 						 *)
	ParamTP_RampQ			: REAL; 		(* (s) Duration for the active power to reach the new setpoint                 						 *)
	                		        		
	//Temp          		        		
	MesTempExt				: REAL;			(* (C°) External temperature *)
			
END_STRUCT
END_TYPE

// ---- 01_Equipement_Library/Inverter/INV_SmaSCXXXXUP_US.TcDUT
TYPE INV_SmaSCXXXXUP_US :
	//SMA CP, CP-US, CP-JP and HE-20
STRUCT
MesData					: INV;

// Device Family
MesIdc_Group1				:REAL; (* (A) DC current inverter bridge 1 [DcMs.Amp.Stk1] *)
MesIdc_Group2				:REAL; (* (A) DC current inverter bridge 2 [DcMs.Amp.Stk2] *)
MesIdc_Group3				:REAL; (* (A) DC current inverter bridge 3 [DcMs.Amp.Stk3] *)
             				
MesUdc_Group1				:REAL; (* (V) DC voltage of the inverter bridge 1 [InvMs.DclVol.Stk1] *)
MesUdc_Group2				:REAL; (* (V) DC voltage of the inverter bridge 2 [InvMs.DclVol.Stk2] *)
MesUdc_Group3				:REAL; (* (V) DC voltage of the inverter bridge 3 [InvMs.DclVol.Stk3] *)
MesI1						:REAL; (* (A) AC current L1, total [InvMs.TotA.PhsA] *)
MesI2						:REAL; (* (A) AC current L2, total [InvMs.TotA.PhsB] *)
MesI3						:REAL; (* (A) AC current L3, total [InvMs.TotA.PhsC] *)

MesU12						:REAL; (* (V) Line-to-line voltage L1-L2, utility grid [GriMs.V.PhsAB] *)
MesU23						:REAL; (* (V) Line-to-line voltage L2-L3, utility grid [GriMs.V.PhsBC] *)
MesU31						:REAL; (* (V) Line-to-line voltage L3-L1, utility grid [GriMs.V.PhsCA] *)

MesTemp_CabAC				:REAL; (* (°C) Temperature in the AC range [TmpCab.Acc] *)
MesTemp_CabDC				:REAL; (* (°C) Temperature in the DC range [TmpCab.Dcc] *)
MesTemp_CabRio				:REAL; (* (°C) Temperature in the electronics area [TmpCab.Rio] *)

MesTemp_Igbt				:REAL; (* (°C) Temperature of the inverter bridge (switch), maximum value [TmpStk.IgbtMax] *)
MesTemp_Pcb					:REAL; (* (°C) Temperature of the inverter bridge (assembly), maximum value [TmpStk.PcbMax] *)
MesTemp_Ext					:REAL; (* (°C) Outside temperature [TmpExl] *)
MesTemp_Transfo				:REAL; (* (°C) Temperature of the MV transformer [TmpTrf] *)
MesID_DC1State				:UINT; (* (-) Switching status of the DC load- break switch 1 [DcSw1Stt] *)
MesID_DC2State				:UINT; (* (-) Switching status of the DC load- break switch 2 [DcSw2Stt] *)
MesID_DC3State				:UINT; (* (-) Switching status of the DC load- break switch 3 [DcSw3Stt] *)
MesID_ACState				:UINT; (* (-) Switching status of the AC circuit breaker [AcSwStt] *)
MesID_CapaState				:UINT; (* (-) Switching state of the capacitor contactor [CapacSwStt] *)
MesID_PreChargeState			:UINT; (* (-) Switching status of the pre-charging contactor [PrchrgSwStt] *)
MesFeedTm					:REAL; (* (s) Feed-in time [Cnt.TotFeedTm] *)
MesWorkingHr				:REAL; (* (s) Operating time [Cnt.TotOpTm] *)
MesEdcDischarge_Tot			:REAL; (* (MWh) DC energy drawn, total [Cnt.TotWatthIn] *)
MesEActProd_Tot				:REAL; (* (MWh) AC energy fed in, total [Cnt.TotWhOut] *)
MesEdcDischarge_Day			:REAL; (* (MWh) DC energy drawn that day [Cnt.WatthIn] *)
MesEActProd_Day				:REAL; (* (MWh) AC energy fed in that day [Cnt.WhOut] *)
MesWorkingHr_Fan1			:REAL; (* (s) Operating time of the interior fan 1 [Cnt.FanCab1Tm] *)
MesWorkingHr_Fan2			:REAL; (* (s) Operating time of the interior fan 2 [Cnt.FanCab2Tm] *)
MesWorkingHr_BridgeFan		:REAL; (* (s) Operating time of the inverter bridge fan [Cnt.FanStkTm] *)
MesWorkingHr_Heater			:REAL; (* (s) Operating time of the interior heater [Cnt.HtCabTm] *)
MesWorkingHr_Heater2		:REAL; (* (s) Operating time of the  -40 C interior heater [Cnt.HtLoExlTmpTm] *)
MesID_ErrorLocation			:UINT; (* (-) Error location of the present error [ErrLcn] *)
MesID_ErrorState			:UINT; (* (-) Error status of the inverter [ErrStt] *)
MesEventID					:REAL; (* (-) Error number of the present error [ErrNo] *)

MesID_StartKeyState			:UINT; (* (-) Switch status of the start-stop key switch [Rio.KeySw] *)
MesTime_GridConnWait		:REAL; (* (s) Waiting time for grid connection [WaitGriTm] *)

MesID_GFDIState				:UINT; (* (-) Switching status of the GFDI [GfdiSwStt] *)
MesSetptP					:REAL; (* (kW) Active power, setpoint [WSpt] *)
MesSetptSmax				:REAL; (* (kVA) Maximum apparent power, setpoint [VAMaxSpt] *)
MesSetptQ					:REAL; (* (kVAr) Reactive power, setpoint [VArSpt] *)
MesSetptCosPhi				:REAL; (* (-) Power factor cos (phi), setpoint [PFSpt] *)
MesID_AlarmGas_Transfo			:UINT; (* (-) Fast stop hermetic protection, pressure [TrfPro.Pres] *)
MesID_AlarmTemp_Transfo		:UINT; (* (-) Fast stop hermetic protection, temperature [TrfPro.TmpTrp] *)
MesID_AlarmOilLevel_Transfo	:UINT; (* (-) Hermetic protection, gas fill level [TrfPro.GasOilLev] *)
MesIDWarningTemp_Transfo		:UINT; (* (-) Hermetic pressure, temperature warning [TrfPro.TmpWrn] *)
MesTemp_Igbt1				:REAL; (* (°C) Temperature of inverter bridge 1 (switch) [TmpStk1.lgbt] *)
MesTemp_Pcb1				:REAL; (* (°C) Maximum temperature of inverter bridge 1 (assembly) [TmpStk1.Pcb] *)
MesTemp_Pcb2				:REAL; (* (°C) Maximum temperature of inverter bridge 2 (assembly) [TmpStk2.Pcb] *)
MesTemp_Pcb3				:REAL; (* (°C) Maximum temperature of inverter bridge 3 (assembly) [TmpStk3.Pcb] *)
MesEAct_PreviousDay			:REAL; (* (MWh) AC energy fed in the previous day [Cnt.YstdWhOut] *)
MesWorkingHr_Cpu			:REAL; (* (s) CPU running time since system start [Cpu1UpTime] *)

MesPressure_Transfo			:REAL; (* (-) MV transformer pressure [PresTrf] *)
MesID_PresMonitorState_Transfo:UINT; (* (-) Error status of MV transformer pressure monitoring [PresTrf.ErrStt] *)
MesState_BackFeedMode		:REAL; (* (-) Status of the function Backfeed Power [BfpBits] *)
MesIdc_BackFeed				:REAL; (* (A) Backfeed Power: DC current used by customer loads [DcMs.BfpAmp] *)

MesEdcCharge_Tot			:REAL; (* (MWh) DC energy fed in, total [Cnt.TotDcWhOut] *)
MesEActCons_Tot				:REAL; (* (MWh) AC energy drawn, total [Cnt.TotAcWhIn] *)
MesEdcCharge_Day			:REAL; (* (MWh) DC energy fed in that day [Cnt.DcWhOut] *)
MesEActCons_Day				:REAL; (* (MWh) AC energy drawn that day [Cnt.AcWhIn] *)
MesSetptUdc					:REAL; (* (V) DC voltage, setpoint [DclVolSpt] *)
MesSetptU					:REAL; (* (pu) AC voltage-dependent reactive power control: setpoint AC voltage [VolNomSpt] *)

MesSetptFreq					:REAL; (* (Hz) Nominal frequency for frequency- dependent control of active power [HzNomSpt] *)
MesPconnected					:REAL; (* (pu) Currently available active power [WAval] *)
MesQconnected					:REAL; (* (pu) Currently available reactive power [VArAval] *)
MesID_Derating				:UINT; (* (-) Current derating status [DrtStt] *)
MesID_Off					:UINT; (* (-) Current cause of inverter disconnection [PwrOffReas] *)
MesTime_SelfTestWait		:REAL; (* (s) Time until the next inverter self test [DiagRmgTm] *)
MesID_WarningFloatCtrl		:REAL; (* (-) The float controller indicates a warning. [Rio.Din.FloatCtl.Wa rn] *)
MesID_ErrorFloatCtrl		:REAL; (* (-) The float controller indicates a warning. [Rio.Din.FloatCtl.Err] *)
MesIGnd						:REAL; (* (A) Ground current measured at the GFDI [Gfdi.AmpPrc] *)
MesIGnd_LastError			:REAL; (* (A) Last measured ground current in case of an error [Gfdi.AmpErr] *)
MesEventID1					:REAL; (* (-) Error number of the current error [ActErrNo1] *)
MesID_ErrorLocation1		:UINT; (* (-) Location where the current error was detected [ActErrLcn1] *)
MesEventID2					:REAL; (* (-) Error number of the current error [ActErrNo2] *)
MesID_ErrorLocation2		:UINT; (* (-) Location where the current error was detected [ActErrLcn2] *)
MesEventID3					:REAL; (* (-) Error number of the current error [ActErrNo3] *)
MesID_ErrorLocation3		:UINT; (* (-) Location where the current error was detected [ActErrLcn3] *)
MesEventID4					:REAL; (* (-) Error number of the current error [ActErrNo4] *)
MesID_ErrorLocation4		:UINT; (* (-) Location where the current error was detected [ActErrLcn4] *)
MesEventID5					:REAL; (* (-) Error number of the current error [ActErrNo5] *)
MesID_ErrorLocation5		:UINT; (* (-) Location where the current error was detected [ActErrLcn5] *)
MesEventID6					:REAL; (* (-) Error number of the current error [ActErrNo6] *)
MesID_ErrorLocation6		:UINT; (* (-) Location where the current error was detected [ActErrLcn6] *)
MesEventID7					:REAL; (* (-) Error number of the current error [ActErrNo7] *)
MesID_ErrorLocation7		:UINT; (* (-) Location where the current error was detected [ActErrLcn7] *)
MesEventID8					:REAL; (* (-) Error number of the current error [ActErrNo8] *)
MesID_ErrorLocation8		:UINT; (* (-) Location where the current error was detected [ActErrLcn8] *)
MesEventID9					:REAL; (* (-) Error number of the current error [ActErrNo9] *)
MesID_ErrorLocation9		:UINT; (* (-) Location where the current error was detected [ActErrLcn9] *)
MesEventID10				:UINT; (* (-) Error number of the current error [ActErrNo10] *)
MesID_ErrorLocation10		:UINT; (* (-) Location where the current error was detected [ActErrLcn10] *)

	
MesIdc_input1			:REAL; (* (A) DC current input X61 [DcMs.Amp.01] *)
MesIdc_input2			:REAL; (* (A) DC current input X62[DcMs.Amp.02] *)
MesIdc_input3			:REAL; (* (A) DC current input X63[DcMs.Amp.03] *)
MesIdc_input4			:REAL; (* (A) DC current input X64[DcMs.Amp.04] *)
MesIdc_input5			:REAL; (* (A) DC current input X65[DcMs.Amp.05] *)
MesIdc_input6			:REAL; (* (A) DC current input X66[DcMs.Amp.06] *)
MesIdc_input7			:REAL; (* (A) DC current input X67[DcMs.Amp.07] *)
//MesIdc_input8			:REAL; (* (A) DC current input X68[DcMs.Amp.08] *)
MesIdc_input9			:REAL; (* (A) DC current input X69[DcMs.Amp.09] *)
MesIdc_input10			:REAL; (* (A) DC current input X70 [DcMs.Amp.10] *)
MesIdc_input11			:REAL; (* (A) DC current input X71 [DcMs.Amp.11] *)
MesIdc_input12			:REAL; (* (A) DC current input X72 [DcMs.Amp.12] *)
MesIdc_input13			:REAL; (* (A) DC current input X73 [DcMs.Amp.13] *)
MesIdc_input14			:REAL; (* (A) DC current input X74 [DcMs.Amp.14] *)
MesIdc_input15			:REAL; (* (A) DC current input X75 [DcMs.Amp.15] *)
//MesIdc_input16			:REAL; (* (A) DC current input X76 [DcMs.Amp.16] *)
MesIdc_input17			:REAL; (* (A) DC current input X77[DcMs.Amp.01] *)
MesIdc_input18			:REAL; (* (A) DC current input X78 [DcMs.Amp.02] *)
MesIdc_input19			:REAL; (* (A) DC current input X79 [DcMs.Amp.03] *)
MesIdc_input20			:REAL; (* (A) DC current input X80 [DcMs.Amp.04] *)
MesIdc_input21			:REAL; (* (A) DC current input X81 [DcMs.Amp.05] *)
MesIdc_input22			:REAL; (* (A) DC current input X82 [DcMs.Amp.06] *)
MesIdc_input23			:REAL; (* (A) DC current input X83 [DcMs.Amp.07] *)
//MesIdc_input24			:REAL; (* (A) DC current input 84 [DcMs.Amp.08] *)



MesStatus_Derating				:WORD; (* (-) Internal Current derating status [DrtStt] *)
MesStatus_Derating1				:WORD; (* (-) Internal Current derating status [DrtStt] *)
MesStatus_Off					:WORD; (* (-) Internal Current cause of inverter disconnection [PwrOffReas] *)
MesStatus_Off1					:WORD; (* (-) Internal Current cause of inverter disconnection [PwrOffReas] *)
		
	
END_STRUCT
END_TYPE

// ---- 01_Equipement_Library/Inverter/JuncBox.TcDUT
TYPE JuncBox :
STRUCT
	/// STR 
	AX_STR: ARRAY[1..CstNbSTR_SB_G] OF STR_SSM;

	MesClosed_DCSwitch	: BOOL ; // State of DC Switch 

	/// Status of signal contact 1 [Signal contact 1]: 303 =Off , 308 = On
	MesID_SignalContact1: WORD;
	/// Status of signal contact 2 [Signal contact 2]: 303 =Off , 308 = On
	MesID_SignalContact2: WORD;
END_STRUCT
END_TYPE

// ---- 01_Equipement_Library/Inverter/PowerCol_INV_Jema.TcDUT
TYPE PowerCol_INV_Jema :
STRUCT
	
	MesData				: PowerCol_INV ; 
	
	MesTempControl  	: REAL; 	(* (°C) Temperature of control card*)
	MesIn_State			: WORD;     (* (NA) MesIn_State		*)
	MesOut_State		: WORD;     (* (NA) MesOut_State	*)
	MesTempPowerUnit	: REAL;     (* (NA) MesTempPowerUnit*)
	MesTempCabinet		: REAL;     (* (NA) MesTempCabinet	*)
	MesRegAlarm0		: WORD;     (* (NA) MesRegAlarm0	*)
	MesRegAlarm1		: WORD;     (* (NA) MesRegAlarm1	*)
	MesRegAlarm2		: WORD;     (* (NA) MesRegAlarm2	*)
	MesRegAlarm3		: WORD;     (* (NA) MesRegAlarm3	*)
	MesRegAlarm4		: WORD;     (* (NA) MesRegAlarm4	*)
	MesDeratingWord		: WORD ;	(*	(NA) Derating word of PCS*)
	MesHeartbit			: REAL ;	(*	(NA) Heartbit*)
	MesDoorOpened		: BOOL ;	(*	(NA) Door of the Power module is opened	*)
		
	MesJemaAlarms		: PowerCol_INV_JemaAlarms; (* Alarms Struct*)
	

END_STRUCT
END_TYPE

// ---- 01_Equipement_Library/Inverter/PowerCol_INV_JemaAlarms.TcDUT
TYPE PowerCol_INV_JemaAlarms :
STRUCT

// ALARM0 bAlarm1
		MesI1_Alm				: BOOL; 	//RegAlarms0: I1_Alm
		MesI2_Alm				: BOOL; 	//RegAlarms0: I2_Alm
		MesI3_Alm				: BOOL; 	//RegAlarms0: I3_Alm
		MesVdc_High_Alm			: BOOL; 	//RegAlarms0: Vdc_High_Alm
		MesVdc_Low_Alm			: BOOL; 	//RegAlarms0: Vdc_Low_Alm
		                    	        	// 
		MesU12_High_Alm			: BOOL; 	//RegAlarms0: U12_High_Alm
		MesU12_Low_Alm			: BOOL; 	//RegAlarms0: U12_Low_Alm
		MesU23_High_Alm			: BOOL; 	//RegAlarms0: U23_High_Alm
		MesU23_Low_Alm			: BOOL; 	//RegAlarms0: U23_Low_Alm
		MesU31_High_Alm			: BOOL; 	//RegAlarms0: U31_High_Alm
		MesU31_Low_Alm			: BOOL; 	//RegAlarms0: U31_Low_Alm
		MesVd_High_Alm			: BOOL; 	//RegAlarms0: Vd_High_Alm
		MesVd_Low_Alm			: BOOL; 	//RegAlarms0: Vd_Low_Alm
		MesVdc_Neg				: BOOL; 	//RegAlarms0: Vdc_Neg
		MesIdc_Neg				: BOOL;		//RegAlarms0: Idc_Neg
											//MesAlarm0
		                    	
// ALARM1 bAlarm1           	
		MesU1223_Unbalance		: BOOL;		//RegAlarms1: U1223_Unbalance
		MesU2331_Unbalance		: BOOL;		//RegAlarms1: U2331_Unbalance
		MesU3112_Unbalance		: BOOL;		//RegAlarms1: U3112_Unbalance
		MesInvertedPhase		: BOOL;		//RegAlarms1: InvertedPhase
		MesI12_Unbalance		: BOOL;		//RegAlarms1: I12_Unbalance
		MesI23_Unbalance		: BOOL;		//RegAlarms1: I23_Unbalance
		MesI31_Unbalance		: BOOL;		//RegAlarms1: I31_Unbalance
											//
		MesF_High				: BOOL;		//RegAlarms1: F_High
		MesF_Low				: BOOL;		//RegAlarms1: F_Low
											//
											//
		MesPcbOverTemp			: BOOL;		//RegAlarms1: PcbOverTemp
		//wAlarmCode
// ALARM2 bAlarm1
											// 
                                    		// 
                                    		// 
                                    		// 
		MesGridCbOpened			: BOOL;		//RegAlarms2: GridCbOpened
		MesGridCbTrip			: BOOL;		//RegAlarms2: GridCbTrip
											//
		                    	       		// 
		MesGridContactFail		: BOOL;		//RegAlarms2: GridContactFail 
		MesDoorOpened			: BOOL;		//RegAlarms2: DoorOpened 
		                    	       		// 
		                    	       		// 
		                    	       		// 
		MesAuxCbOpened			: BOOL;		//RegAlarms2: AuxCbOpened 
		MesOverVoltHyst			: BOOL;		//RegAlarms2: OverVoltHyst 
		MesIdcMax				: BOOL;		//RegAlarms2: IdcMax 
		//wAlarmCode
		
//ALARM3   bAlarm1                         
		MesSKIIP1				: BOOL; 	//RegAlarms3: SKIIP1
		MesSKIIP2				: BOOL; 	//RegAlarms3: SKIIP2
		MesSKIIP3				: BOOL; 	//RegAlarms3: SKIIP3
		MesSKIIP_OT				: BOOL; 	//RegAlarms3: SIIP_OT
		MesHardwareOverCurrent	: BOOL; 	//RegAlarms3: FPGA_WdogTrip
		MesStopEverything		: BOOL; 	//RegAlarms3: StopEverything
		MesIMax					: BOOL; 	//RegAlarms3: IMax
		MesEmergencyStop		: BOOL; 	//RegAlarms3: EmergencyStop
		MesImdWarning			: BOOL; 	//RegAlarms3: ImdWarning
		MesImdFault				: BOOL; 	//RegAlarms3: ImdFault
		                    	        	//RegAlarms3:  
		MesCoilOverTemp			: BOOL; 	//RegAlarms3: CoilOverTemp
		                    	        	//RegAlarms3:  
		MesAlrmGrp1_Curr		: BOOL; 	//RegAlarms3: AlrmGrp1_Curr
		MesAlrmGrp2_Curr		: BOOL; 	//RegAlarms3: AlrmGrp2_Curr
		MesShortCircuit_DC		: BOOL; 	//RegAlarms3: ShortCircuit_DC
		//wAlarmCode		
		
	//Input1                		
		Es							: BOOL; // Emergency Stop 
		DsAc						: BOOL;	// AC Door Open 
		AcSurge						: BOOL;	// FeedBack Parafoudre AC Burned
		GridCircuitBreakerDrop		: BOOL; // Circuit Breaker DC Open ??
		VaristorProtCabAux			: BOOL; // Varistor protection cabinet auxiliaire
		PlcOverTemp					: BOOL;	// Warning not alarms : Temp PLC under 40°
		UnderTemp					: BOOL; // Low temperature, under 5°
		Humidity					: BOOL;	// Humidity
		Es_Or_CbDcOpen				: BOOL;	// Emergy Stop or circuit breaker dc open
		
	//Input2
		CB_Motor1_Closed			: BOOL;	// Sectionneur DC 1 fermé
		CB_Motor2_Closed			: BOOL;	// Sectionneur DC 1 fermé
		CB_Motor3_Closed			: BOOL;	// Sectionneur DC 1 fermé
		Ground_Fault_Lvl1_Bender	: BOOL; // Warning Lvl 1 ground fault from bender
		Ground_Fault_Lvl2_Bender	: BOOL; // Alarms  Lvl 2 ground fault from bender
		DsDc						: BOOL;	// Porte gauche fermé
		DsSafe						: BOOL;	// Porte droite fermé
		DcSurge						: BOOL; // FeedBack DC Surge
		HeatingFail					: BOOL; // Error on heating system
		CapaDischarge				: BOOL; // IS discharging Capacity
		GFDI_Close					: BOOL;	// GFDHI IS CLOSE
		GFDI_Open					: BOOL;	// GFDI IS OPEN
		GFDI_Trip					: BOOL;	// GFDI HAS TRIPPED
END_STRUCT
END_TYPE

// ---- 01_Equipement_Library/Inverter/PowerCol_INV.TcDUT
TYPE PowerCol_INV :
STRUCT
	MesUdc 				: REAL;  	(* (V) DC Voltage measure*)
	MesIdc 				: REAL; 	(* (A) Total DC current from batteries (+ = discharge)*)
	MesV1 				: REAL;  	(* (V) AC Voltage measure*)
	MesV2				: REAL;     (* (V) AC Voltage measure*)
	MesV3				: REAL;     (* (V) AC Voltage measure*)
	MesI1				: REAL; 	(* (A) Phase 1 AC Current*)
	MesI2				: REAL;     (* (A) Phase 2 AC Current*)
	MesI3				: REAL;     (* (A) Phase 3 AC Current*)
	MesPdc				: REAL; 	(* (kW) DC Power . *)
	MesP 				: REAL; 	(* (kW) Active Power output (AC) of PCS*)
	MesQ 				: REAL; 	(* (kVAr) Reactive AC Power Produced by PCS *)
	MesCosPhi 			: REAL;  	(* (p.u) Power factor*)
	MesFreq				: REAL; 	(* (Hz) Frequency*)
	MesAcSwitchClosed	: BOOL ; 	(*NA) Position of the AC Switch : True = Switch closed*)

	MesAlarmCode		: WORD ; 		(* (NA) 	Internal Akuo AlarmCode         *)             															
	MesWarningCode		: WORD ; 		(* (NA) 	Internal Akuo WarningCode       *)             															
	MesEventCode		: WORD ; 		(* (NA) 	Internal Akuo EventCode         *)
	
	
END_STRUCT
END_TYPE

// ---- 01_Equipement_Library/Inverter/PowerCol_INV_Power_One.TcDUT
TYPE PowerCol_INV_Power_One :


STRUCT
	

			MesData			: PowerCol_INV ; 
			
		//INV Caracteristiques
			MesSN				: UINT;      (*  		Serial Number*)
			MesID_Type			: UINT; 		(*          0=Master MPPT 1=slave MPTT*)
			MesID_StateGlobal	: UINT;      (*			Global state, Note 2.1*)
			MesIDState			: UINT;      (*			Inverter State, Note 2.2  *)
			MesAlarmID			: UINT;      (*          Alarm state, Note2.4*)
		// INV Measures
			MesEDay				: REAL;     (* (kWh)	Daily Energy*)
			MesETot				: REAL;		(* (kWh)    Total Energy*)
			MesEPartial			: REAL;		(* (kWh)	??? To check*)
			MesEWeek			: REAL;		(* (kWh)	Week Energy*)
			MesEMonth			: REAL;		(* (kWh)	Monthly Energy*)
			MesEYear			: REAL;     (* (kWh)	Yearly Energy*)
			
			MesV				: REAL;		(* (V)		Average 3 phases Grid Volatage For Slave*)
			MesI		 		: REAL;  	(* (A) 		Average 3 phases Grid Current For Slave*)
		 
			MesTemp_Inv			: REAL;		(* (°C)		Supervisor Temperature*)
			MesTemp_Supply			: REAL;		(* (°C)		Power Supply Temperature*)
			MesTemp_Headsink			: REAL;		(* (°C)		Headsink*)
			MesTemp_T2					: REAL;		(* (°C)		T2*)
			MesTemp_T3					: REAL; 	(* (°C)		T3*)
	
END_STRUCT
END_TYPE

// ---- 01_Equipement_Library/Inverter/INV_Huawei_SL.TcDUT
///////////
// Structure For Inverter. Main Operating Data to be saved ( ex: OPC ) .  
//////////
TYPE INV_Huawei_SL :
STRUCT
	
		MesData				: INV ;  (* INV *) 
	
	// INV Measures
		MesEDay				: REAL ;     	(*/ (kWh) Daily Energy*)
	    MesETot				: REAL ;		(*/ (kWh) Total Energy*)
		MesOn				: BOOL ;        (* Smartlogger is ON*)
		MesI1				: REAL ;        (* (A) AC current phase 1*)
		MesI2				: REAL ;        (* (A) AC current phase 1*)
	    MesI3				: REAL ;        (* (A) AC current phase 1*)
		MesU12				: REAL ;        (*(V) AC Voltage phase1 to phase2*)
        MesU23				: REAL ;        (*(V) AC Voltage phase2 to phase3*)
        MesU31				: REAL ;        (*(V) AC Voltage phase3 to phase1*)
		MesEff				: REAL ; 		(* (%) Inverter efficiency*)
		MesSetptPMax		: REAL ;        (* (kW) Maximal Active power setpoint*)
		MesSetptQMax		: REAL ;        (*(kVAr) Maximal reactive power setpoint*)
		MesSetptQMin		: REAL ;        (*(kVAr) Minimal reactive power setpoint*)
		OUT_SetptPlimit		: REAL ;        (*(kW) Maximal Active power setpoint sent by PPC*)
		OUT_SetptQlimit		: REAL ;        (*(kVAr) Maximal Reactive power setpoint sent by PPC*)

END_STRUCT
END_TYPE

// ---- 01_Equipement_Library/Inverter/STR.TcDUT
TYPE STR :
STRUCT
		MesIdc			: REAL;   						(* (A) DC current *)
		MesUdc			: REAL;							(* (V) DC voltage *)
END_STRUCT
END_TYPE

// ---- 01_Equipement_Library/Inverter/STR_SSM.TcDUT
TYPE STR_SSM :
STRUCT
		MesData			: STR ; 


		MesPdc				: REAL ; (* (A) DC Power *)
(*		MesIdc_1			: REAL;   						(* (A) DC current *)
		MesIdc_2			: REAL;   						(* (A) DC current *)
		MesIdc_3			: REAL;   						(* (A) DC current *)
		MesIdc_4			: REAL;   						(* (A) DC current *)
		MesIdc_5			: REAL;   						(* (A) DC current *)
		MesIdc_6			: REAL;   						(* (A) DC current *)
		MesIdc_7			: REAL;   						(* (A) DC current *)
		MesIdc_8			: REAL;   						(* (A) DC current *)		
		
		MesPdc				: REAL ; (* (A) DC Power *)	 *)
END_STRUCT
END_TYPE
(*
AX_PTR[1].AX_INV[2].BJMonitor[1].STR[1]. MesIdc_1
AX_PTR[1].AX_INV[2].BJMonitor[1].STR[1]. MesIdc_2
AX_PTR[1].AX_INV[2].BJMonitor[1].STR[1]. MesIdc_3
AX_PTR[1].AX_INV[2].BJMonitor[1].STR[1]. MesIdc_4
AX_PTR[1].AX_INV[2].BJMonitor[1].STR[1]. MesIdc_5
AX_PTR[1].AX_INV[2].BJMonitor[1].STR[1]. MesIdc_6
AX_PTR[1].AX_INV[2].BJMonitor[1].STR[1]. MesIdc_7
AX_PTR[1].AX_INV[2].BJMonitor[1].STR[1]. MesIdc_8
AX_PTR[1].AX_INV[2].BJMonitor[1].STR[1]. MesPdc
AX_PTR[1].AX_INV[2].BJMonitor[1].STR[2]. MesIdc_1
AX_PTR[1].AX_INV[2].BJMonitor[1].STR[2]. MesIdc_2
AX_PTR[1].AX_INV[2].BJMonitor[1].STR[2]. MesIdc_3
AX_PTR[1].AX_INV[2].BJMonitor[1].STR[2]. MesIdc_4
AX_PTR[1].AX_INV[2].BJMonitor[1].STR[2]. MesIdc_5
AX_PTR[1].AX_INV[2].BJMonitor[1].STR[2]. MesIdc_6
AX_PTR[1].AX_INV[2].BJMonitor[1].STR[2]. MesIdc_7
AX_PTR[1].AX_INV[2].BJMonitor[1].STR[2]. MesIdc_8
AX_PTR[1].AX_INV[2].BJMonitor[1].STR[2]. MesPdc
AX_PTR[1].AX_INV[2].BJMonitor[1].STR[3]. MesIdc_1
AX_PTR[1].AX_INV[2].BJMonitor[1].STR[3]. MesIdc_2
AX_PTR[1].AX_INV[2].BJMonitor[1].STR[3]. MesIdc_3
AX_PTR[1].AX_INV[2].BJMonitor[1].STR[3]. MesIdc_4
AX_PTR[1].AX_INV[2].BJMonitor[1].STR[3]. MesIdc_5
AX_PTR[1].AX_INV[2].BJMonitor[1].STR[3]. MesIdc_6
AX_PTR[1].AX_INV[2].BJMonitor[1].STR[3]. MesIdc_7
AX_PTR[1].AX_INV[2].BJMonitor[1].STR[3]. MesIdc_8
AX_PTR[1].AX_INV[2].BJMonitor[1].STR[3]. MesPdc
AX_PTR[1].AX_INV[2].BJMonitor[2].STR[1]. MesIdc_1
AX_PTR[1].AX_INV[2].BJMonitor[2].STR[1]. MesIdc_2
AX_PTR[1].AX_INV[2].BJMonitor[2].STR[1]. MesIdc_3
AX_PTR[1].AX_INV[2].BJMonitor[2].STR[1]. MesIdc_4
AX_PTR[1].AX_INV[2].BJMonitor[2].STR[1]. MesIdc_5
AX_PTR[1].AX_INV[2].BJMonitor[2].STR[1]. MesIdc_6
AX_PTR[1].AX_INV[2].BJMonitor[2].STR[1]. MesIdc_7
AX_PTR[1].AX_INV[2].BJMonitor[2].STR[1]. MesIdc_8
AX_PTR[1].AX_INV[2].BJMonitor[2].STR[1]. MesPdc
AX_PTR[1].AX_INV[2].BJMonitor[2].STR[2]. MesIdc_1
AX_PTR[1].AX_INV[2].BJMonitor[2].STR[2]. MesIdc_2
AX_PTR[1].AX_INV[2].BJMonitor[2].STR[2]. MesIdc_3
AX_PTR[1].AX_INV[2].BJMonitor[2].STR[2]. MesIdc_4
AX_PTR[1].AX_INV[2].BJMonitor[2].STR[2]. MesIdc_5
AX_PTR[1].AX_INV[2].BJMonitor[2].STR[2]. MesIdc_6
AX_PTR[1].AX_INV[2].BJMonitor[2].STR[2]. MesIdc_7
AX_PTR[1].AX_INV[2].BJMonitor[2].STR[2]. MesIdc_8
AX_PTR[1].AX_INV[2].BJMonitor[2].STR[2]. MesPdc
AX_PTR[1].AX_INV[2].BJMonitor[2].STR[3]. MesIdc_1
AX_PTR[1].AX_INV[2].BJMonitor[2].STR[3]. MesIdc_2
AX_PTR[1].AX_INV[2].BJMonitor[2].STR[3]. MesIdc_3
AX_PTR[1].AX_INV[2].BJMonitor[2].STR[3]. MesIdc_4
AX_PTR[1].AX_INV[2].BJMonitor[2].STR[3]. MesIdc_5
AX_PTR[1].AX_INV[2].BJMonitor[2].STR[3]. MesIdc_6
AX_PTR[1].AX_INV[2].BJMonitor[2].STR[3]. MesIdc_7
AX_PTR[1].AX_INV[2].BJMonitor[2].STR[3]. MesIdc_8
AX_PTR[1].AX_INV[2].BJMonitor[2].STR[3]. MesPdc
AX_PTR[1].AX_INV[2].BJMonitor[3].STR[1]. MesIdc_1
AX_PTR[1].AX_INV[2].BJMonitor[3].STR[1]. MesIdc_2
AX_PTR[1].AX_INV[2].BJMonitor[3].STR[1]. MesIdc_3
AX_PTR[1].AX_INV[2].BJMonitor[3].STR[1]. MesIdc_4
AX_PTR[1].AX_INV[2].BJMonitor[3].STR[1]. MesIdc_5
AX_PTR[1].AX_INV[2].BJMonitor[3].STR[1]. MesIdc_6
AX_PTR[1].AX_INV[2].BJMonitor[3].STR[1]. MesIdc_7
AX_PTR[1].AX_INV[2].BJMonitor[3].STR[1]. MesIdc_8
AX_PTR[1].AX_INV[2].BJMonitor[3].STR[1]. MesPdc
AX_PTR[1].AX_INV[2].BJMonitor[3].STR[2]. MesIdc_1
AX_PTR[1].AX_INV[2].BJMonitor[3].STR[2]. MesIdc_2
AX_PTR[1].AX_INV[2].BJMonitor[3].STR[2]. MesIdc_3
AX_PTR[1].AX_INV[2].BJMonitor[3].STR[2]. MesIdc_4
AX_PTR[1].AX_INV[2].BJMonitor[3].STR[2]. MesIdc_5
AX_PTR[1].AX_INV[2].BJMonitor[3].STR[2]. MesIdc_6
AX_PTR[1].AX_INV[2].BJMonitor[3].STR[2]. MesIdc_7
AX_PTR[1].AX_INV[2].BJMonitor[3].STR[2]. MesIdc_8
AX_PTR[1].AX_INV[2].BJMonitor[3].STR[2]. MesPdc
AX_PTR[1].AX_INV[2].BJMonitor[3].STR[3]. MesIdc_1
AX_PTR[1].AX_INV[2].BJMonitor[3].STR[3]. MesIdc_2
AX_PTR[1].AX_INV[2].BJMonitor[3].STR[3]. MesIdc_3
AX_PTR[1].AX_INV[2].BJMonitor[3].STR[3]. MesIdc_4
AX_PTR[1].AX_INV[2].BJMonitor[3].STR[3]. MesIdc_5
AX_PTR[1].AX_INV[2].BJMonitor[3].STR[3]. MesIdc_6
AX_PTR[1].AX_INV[2].BJMonitor[3].STR[3]. MesIdc_7
AX_PTR[1].AX_INV[2].BJMonitor[3].STR[3]. MesIdc_8
AX_PTR[1].AX_INV[2].BJMonitor[3].STR[3]. MesPdc
AX_PTR[1].AX_INV[2].BJMonitor[4].STR[1]. MesIdc_1
AX_PTR[1].AX_INV[2].BJMonitor[4].STR[1]. MesIdc_2
AX_PTR[1].AX_INV[2].BJMonitor[4].STR[1]. MesIdc_3
AX_PTR[1].AX_INV[2].BJMonitor[4].STR[1]. MesIdc_4
AX_PTR[1].AX_INV[2].BJMonitor[4].STR[1]. MesIdc_5
AX_PTR[1].AX_INV[2].BJMonitor[4].STR[1]. MesIdc_6
AX_PTR[1].AX_INV[2].BJMonitor[4].STR[1]. MesIdc_7
AX_PTR[1].AX_INV[2].BJMonitor[4].STR[1]. MesIdc_8
AX_PTR[1].AX_INV[2].BJMonitor[4].STR[1]. MesPdc
AX_PTR[1].AX_INV[2].BJMonitor[4].STR[2]. MesIdc_1
AX_PTR[1].AX_INV[2].BJMonitor[4].STR[2]. MesIdc_2
AX_PTR[1].AX_INV[2].BJMonitor[4].STR[2]. MesIdc_3
AX_PTR[1].AX_INV[2].BJMonitor[4].STR[2]. MesIdc_4
AX_PTR[1].AX_INV[2].BJMonitor[4].STR[2]. MesIdc_5
AX_PTR[1].AX_INV[2].BJMonitor[4].STR[2]. MesIdc_6
AX_PTR[1].AX_INV[2].BJMonitor[4].STR[2]. MesIdc_7
AX_PTR[1].AX_INV[2].BJMonitor[4].STR[2]. MesIdc_8
AX_PTR[1].AX_INV[2].BJMonitor[4].STR[2]. MesPdc
AX_PTR[1].AX_INV[2].BJMonitor[4].STR[3]. MesIdc_1
AX_PTR[1].AX_INV[2].BJMonitor[4].STR[3]. MesIdc_2
AX_PTR[1].AX_INV[2].BJMonitor[4].STR[3]. MesIdc_3
AX_PTR[1].AX_INV[2].BJMonitor[4].STR[3]. MesIdc_4
AX_PTR[1].AX_INV[2].BJMonitor[4].STR[3]. MesIdc_5
AX_PTR[1].AX_INV[2].BJMonitor[4].STR[3]. MesIdc_6
AX_PTR[1].AX_INV[2].BJMonitor[4].STR[3]. MesIdc_7
AX_PTR[1].AX_INV[2].BJMonitor[4].STR[3]. MesIdc_8
AX_PTR[1].AX_INV[2].BJMonitor[4].STR[3]. MesPdc
AX_PTR[1].AX_INV[2].BJMonitor[5].STR[1]. MesIdc_1
AX_PTR[1].AX_INV[2].BJMonitor[5].STR[1]. MesIdc_2
AX_PTR[1].AX_INV[2].BJMonitor[5].STR[1]. MesIdc_3
AX_PTR[1].AX_INV[2].BJMonitor[5].STR[1]. MesIdc_4
AX_PTR[1].AX_INV[2].BJMonitor[5].STR[1]. MesIdc_5
AX_PTR[1].AX_INV[2].BJMonitor[5].STR[1]. MesIdc_6
AX_PTR[1].AX_INV[2].BJMonitor[5].STR[1]. MesIdc_7
AX_PTR[1].AX_INV[2].BJMonitor[5].STR[1]. MesIdc_8
AX_PTR[1].AX_INV[2].BJMonitor[5].STR[1]. MesPdc
AX_PTR[1].AX_INV[2].BJMonitor[5].STR[2]. MesIdc_1
AX_PTR[1].AX_INV[2].BJMonitor[5].STR[2]. MesIdc_2
AX_PTR[1].AX_INV[2].BJMonitor[5].STR[2]. MesIdc_3
AX_PTR[1].AX_INV[2].BJMonitor[5].STR[2]. MesIdc_4
AX_PTR[1].AX_INV[2].BJMonitor[5].STR[2]. MesIdc_5
AX_PTR[1].AX_INV[2].BJMonitor[5].STR[2]. MesIdc_6
AX_PTR[1].AX_INV[2].BJMonitor[5].STR[2]. MesIdc_7
AX_PTR[1].AX_INV[2].BJMonitor[5].STR[2]. MesIdc_8
AX_PTR[1].AX_INV[2].BJMonitor[5].STR[2]. MesPdc
AX_PTR[1].AX_INV[2].BJMonitor[5].STR[3]. MesIdc_1
AX_PTR[1].AX_INV[2].BJMonitor[5].STR[3]. MesIdc_2
AX_PTR[1].AX_INV[2].BJMonitor[5].STR[3]. MesIdc_3
AX_PTR[1].AX_INV[2].BJMonitor[5].STR[3]. MesIdc_4
AX_PTR[1].AX_INV[2].BJMonitor[5].STR[3]. MesIdc_5
AX_PTR[1].AX_INV[2].BJMonitor[5].STR[3]. MesIdc_6
AX_PTR[1].AX_INV[2].BJMonitor[5].STR[3]. MesIdc_7
AX_PTR[1].AX_INV[2].BJMonitor[5].STR[3]. MesIdc_8
AX_PTR[1].AX_INV[2].BJMonitor[5].STR[3]. MesPdc
AX_PTR[1].AX_INV[2].BJMonitor[6].STR[1]. MesIdc_1
AX_PTR[1].AX_INV[2].BJMonitor[6].STR[1]. MesIdc_2
AX_PTR[1].AX_INV[2].BJMonitor[6].STR[1]. MesIdc_3
AX_PTR[1].AX_INV[2].BJMonitor[6].STR[1]. MesIdc_4
AX_PTR[1].AX_INV[2].BJMonitor[6].STR[1]. MesIdc_5
AX_PTR[1].AX_INV[2].BJMonitor[6].STR[1]. MesIdc_6
AX_PTR[1].AX_INV[2].BJMonitor[6].STR[1]. MesIdc_7
AX_PTR[1].AX_INV[2].BJMonitor[6].STR[1]. MesIdc_8
AX_PTR[1].AX_INV[2].BJMonitor[6].STR[1]. MesPdc
AX_PTR[1].AX_INV[2].BJMonitor[6].STR[2]. MesIdc_1
AX_PTR[1].AX_INV[2].BJMonitor[6].STR[2]. MesIdc_2
AX_PTR[1].AX_INV[2].BJMonitor[6].STR[2]. MesIdc_3
AX_PTR[1].AX_INV[2].BJMonitor[6].STR[2]. MesIdc_4
AX_PTR[1].AX_INV[2].BJMonitor[6].STR[2]. MesIdc_5
AX_PTR[1].AX_INV[2].BJMonitor[6].STR[2]. MesIdc_6
AX_PTR[1].AX_INV[2].BJMonitor[6].STR[2]. MesIdc_7
AX_PTR[1].AX_INV[2].BJMonitor[6].STR[2]. MesIdc_8
AX_PTR[1].AX_INV[2].BJMonitor[6].STR[2]. MesPdc
AX_PTR[1].AX_INV[2].BJMonitor[6].STR[3]. MesIdc_1
AX_PTR[1].AX_INV[2].BJMonitor[6].STR[3]. MesIdc_2
AX_PTR[1].AX_INV[2].BJMonitor[6].STR[3]. MesIdc_3
AX_PTR[1].AX_INV[2].BJMonitor[6].STR[3]. MesIdc_4
AX_PTR[1].AX_INV[2].BJMonitor[6].STR[3]. MesIdc_5
AX_PTR[1].AX_INV[2].BJMonitor[6].STR[3]. MesIdc_6
AX_PTR[1].AX_INV[2].BJMonitor[6].STR[3]. MesIdc_7
AX_PTR[1].AX_INV[2].BJMonitor[6].STR[3]. MesIdc_8
AX_PTR[1].AX_INV[2].BJMonitor[6].STR[3]. MesPdc
AX_PTR[1].AX_INV[2].BJMonitor[7].STR[1]. MesIdc_1
AX_PTR[1].AX_INV[2].BJMonitor[7].STR[1]. MesIdc_2
AX_PTR[1].AX_INV[2].BJMonitor[7].STR[1]. MesIdc_3
AX_PTR[1].AX_INV[2].BJMonitor[7].STR[1]. MesIdc_4
AX_PTR[1].AX_INV[2].BJMonitor[7].STR[1]. MesIdc_5
AX_PTR[1].AX_INV[2].BJMonitor[7].STR[1]. MesIdc_6
AX_PTR[1].AX_INV[2].BJMonitor[7].STR[1]. MesIdc_7
AX_PTR[1].AX_INV[2].BJMonitor[7].STR[1]. MesIdc_8
AX_PTR[1].AX_INV[2].BJMonitor[7].STR[1]. MesPdc
AX_PTR[1].AX_INV[2].BJMonitor[7].STR[2]. MesIdc_1
AX_PTR[1].AX_INV[2].BJMonitor[7].STR[2]. MesIdc_2
AX_PTR[1].AX_INV[2].BJMonitor[7].STR[2]. MesIdc_3
AX_PTR[1].AX_INV[2].BJMonitor[7].STR[2]. MesIdc_4
AX_PTR[1].AX_INV[2].BJMonitor[7].STR[2]. MesIdc_5
AX_PTR[1].AX_INV[2].BJMonitor[7].STR[2]. MesIdc_6
AX_PTR[1].AX_INV[2].BJMonitor[7].STR[2]. MesIdc_7
AX_PTR[1].AX_INV[2].BJMonitor[7].STR[2]. MesIdc_8
AX_PTR[1].AX_INV[2].BJMonitor[7].STR[2]. MesPdc
AX_PTR[1].AX_INV[2].BJMonitor[7].STR[3]. MesIdc_1
AX_PTR[1].AX_INV[2].BJMonitor[7].STR[3]. MesIdc_2
AX_PTR[1].AX_INV[2].BJMonitor[7].STR[3]. MesIdc_3
AX_PTR[1].AX_INV[2].BJMonitor[7].STR[3]. MesIdc_4
AX_PTR[1].AX_INV[2].BJMonitor[7].STR[3]. MesIdc_5
AX_PTR[1].AX_INV[2].BJMonitor[7].STR[3]. MesIdc_6
AX_PTR[1].AX_INV[2].BJMonitor[7].STR[3]. MesIdc_7
AX_PTR[1].AX_INV[2].BJMonitor[7].STR[3]. MesIdc_8
AX_PTR[1].AX_INV[2].BJMonitor[7].STR[3]. MesPdc

(*
AX_PTR[1].AX_INV[1].BJMonitor[1].STR[1].MesComError
AX_PTR[1].AX_INV[1].BJMonitor[1].STR[2].MesComError
AX_PTR[1].AX_INV[1].BJMonitor[1].STR[3].MesComError
AX_PTR[1].AX_INV[1].BJMonitor[2].STR[1].MesComError
AX_PTR[1].AX_INV[1].BJMonitor[2].STR[2].MesComError
AX_PTR[1].AX_INV[1].BJMonitor[2].STR[3].MesComError
AX_PTR[1].AX_INV[1].BJMonitor[3].STR[1].MesComError
AX_PTR[1].AX_INV[1].BJMonitor[3].STR[2].MesComError
AX_PTR[1].AX_INV[1].BJMonitor[3].STR[3].MesComError
AX_PTR[1].AX_INV[1].BJMonitor[4].STR[1].MesComError
AX_PTR[1].AX_INV[1].BJMonitor[4].STR[2].MesComError
AX_PTR[1].AX_INV[1].BJMonitor[4].STR[3].MesComError
AX_PTR[1].AX_INV[1].BJMonitor[5].STR[1].MesComError
AX_PTR[1].AX_INV[1].BJMonitor[5].STR[2].MesComError
AX_PTR[1].AX_INV[1].BJMonitor[5].STR[3].MesComError
AX_PTR[1].AX_INV[1].BJMonitor[6].STR[1].MesComError
AX_PTR[1].AX_INV[1].BJMonitor[6].STR[2].MesComError
AX_PTR[1].AX_INV[1].BJMonitor[6].STR[3].MesComError
AX_PTR[1].AX_INV[1].BJMonitor[7].STR[1].MesComError
AX_PTR[1].AX_INV[1].BJMonitor[7].STR[2].MesComError
AX_PTR[1].AX_INV[1].BJMonitor[7].STR[3].MesComError
*)
AX_PTR[2].AX_INV[1].IN_MesClosed_BJ_IO[1]
AX_PTR[2].AX_INV[1].IN_MesClosed_BJ_IO[2]
AX_PTR[2].AX_INV[1].IN_MesClosed_BJ_IO[3]
AX_PTR[2].AX_INV[1].IN_MesClosed_BJ_IO[4]
AX_PTR[2].AX_INV[1].IN_MesClosed_BJ_IO[5]
AX_PTR[2].AX_INV[1].IN_MesClosed_BJ_IO[6]
AX_PTR[2].AX_INV[1].IN_MesClosed_BJ_IO[7]
AX_PTR[2].AX_INV[2].IN_MesClosed_BJ_IO[1]
AX_PTR[2].AX_INV[2].IN_MesClosed_BJ_IO[2]
AX_PTR[2].AX_INV[2].IN_MesClosed_BJ_IO[3]
AX_PTR[2].AX_INV[2].IN_MesClosed_BJ_IO[4]
AX_PTR[2].AX_INV[2].IN_MesClosed_BJ_IO[5]
AX_PTR[2].AX_INV[2].IN_MesClosed_BJ_IO[6]
AX_PTR[2].AX_INV[2].IN_MesClosed_BJ_IO[7]


*)

// ---- 01_Equipement_Library/IPC/IPC.TcDUT
TYPE IPC:
STRUCT
	MesAlarmCode		: WORD;	(* (NA) Internal Akuo AlarmCode  *)
	MesWarningCode		: WORD; (* (NA) Internal Akuo WarningCode*)
	MesEventCode		: WORD; (* (NA) Internal Akuo EventCode	 *)
END_STRUCT
END_TYPE

// ---- 01_Equipement_Library/IPC/IPC_Standard.TcDUT
TYPE IPC_Standard:
STRUCT
	MesData	: IPC;  (* (NA) Object	*)
END_STRUCT
END_TYPE

// ---- 01_Equipement_Library/Operation Meter/PM.TcDUT
///////////
// Structure For I35. Main Operating Data to be saved (ex: OPC).  
//////////
TYPE PM :
STRUCT
		MesU12						: REAL ; (* (V) Phase1 - Phase 2 AC Voltage 		   			*)
		MesU23						: REAL ; (* (V) Phase2 - Phase 3 AC Voltage         			*)
		MesU31						: REAL ; (* (V) Phase3 - Phase 1 AC Voltage         			*)
  		MesV1						: REAL ; (* (V) Phase1 AC Voltage                   			*)
		MesV2						: REAL ; (* (V) Phase2 AC Voltage                   			*)
		MesV3						: REAL ; (* (V) Phase3 AC Voltage		           				*)
		MesFreq						: REAL ; (* (Hz)Frequency		                   				*)
		MesI1						: REAL ; (* (A) AC current Phase 1                  			*)
		MesI2						: REAL ; (* (A) AC current Phase 2                  			*)
		MesI3						: REAL ; (* (A) AC current Phase 3                  			*)
		MesIn						: REAL ; (* (A) Neutral AC current                  			*)
		MesP						: REAL ; (* (kW) Total Active power                 			*)
		MesQ						: REAL ; (* (kVAr) Total Reactive Power Phase 1     			*)
		MesS						: REAL ; (* (kVA)Total Apparent power		       				*)
		MesCosPhi					: REAL ; (* (NA) Power factor                       			*)
		MesP1						: REAL ; (* (kW) Active Power Phase 1               			*)
		MesP2						: REAL ; (* (kW) Active Power Phase 2               			*)
		MesP3						: REAL ; (* (kW) Active Power phase 3               			*)
		MesQ1						: REAL ; (* (kVAr)Reactive Power Phase 1            			*)
		MesQ2						: REAL ; (* (kVAr)Reactive Power Phase 2            			*)
		MesQ3						: REAL ; (* (kVAr)Reactive Power Phase 3            			*)
		MesS1						: REAL ; (* (kVA) Total Apparent power Phase 1      			*)
		MesS2						: REAL ; (* (kVA) Total Apparent power Phase 2      			*)
		MesS3						: REAL ; (* (kVA) Total Apparent power Phase 3      			*)
		MesEActCons					: REAL ; (* (kWh) Recieved active energy            			*)
		MesEReactCons				: REAL ; (* (kVArh) 	Recieved reactive energy       			*)
		MesEActProd					: REAL ; (* (kWh) Delivered active energy           			*)
		MesEReactProd				: REAL ; (* (kVArh) 	Delivered reactive energy	   			*)
		MesI						: REAL ; (* (A) Mean AC current                     			*)
		MesV						: REAL ; (* (V) Mean Simple Phase AC Voltage        			*)
		MesU						: REAL ; (* (V) Mean Phase - Phase  AC Voltage      			*)
		MesCosPhi1                  : REAL ; (* (NA) Total Power Factor Phase 1         			*)
		MesCosPhi2                  : REAL ; (* (NA) Total Power Factor Phase 2         			*)
		MesCosPhi3                  : REAL ; (* (NA) Total Power Factor Phase 3         			*)
		MesTanPhi					: REAL ; (* (NA) Total Tangeante phi                			*)

		MesAlarmCom					: BOOL ;  		 (* (NA) Communication Error with I35 module    *)
		MesCP_Read					: BOOL := TRUE ; (* (NA) Cal: Read FUNCTION enable 				*)
		                                                                                        	
		MesAlarmCode				: WORD ; (* (NA) Internal Akuo Alarm Code			   			*)
		MesWarningCode				: WORD ; (* (NA) Internal Akuo Warning Code			  			*)
END_STRUCT
END_TYPE

// ---- 01_Equipement_Library/Operation Meter/PM_DirisA40.TcDUT
///////////
// Structure For I35. Main Operating Data to be saved (ex: OPC).  
//////////
TYPE PM_DirisA40 :
STRUCT
		MesData						: PM ; (* Object *) 
		
		
		MesComAlarm		: BOOL ;			(* (NA) Akuo Com Alarm*)
		MesComWarning	: BOOL ;			(* (NA) Akuo Com Warning*)
		MesTHDU12		: REAL ; 			(* (%) THD *)
		MesTHDU23       : REAL ;            (* (%) THD *)
		MesTHDU31       : REAL ;            (* (%) THD *)
		MesTHDV1        : REAL ;            (* (%) THD *)
		MesTHDV2        : REAL ;            (* (%) THD *)
		MesTHDV3        : REAL ;            (* (%) THD *)
		MesTHDI1        : REAL ;            (* (%) THD *)
		MesTHDI2        : REAL ;            (* (%) THD *)
		MesTHDI3        : REAL ;            (* (%) THD *)
		MesTHDIN        : REAL ;            (* (%) THD *)
		
		
END_STRUCT
END_TYPE

// ---- 01_Equipement_Library/Operation Meter/PM_ION9200.TcDUT
///////////
// Structure For I35. Main Operating Data to be saved (ex: OPC).  
//////////
TYPE PM_ION9200 :
STRUCT
		MesData						: PM ; (* Object *) 
		MesSeconds					: REAL;
		
		
END_STRUCT
END_TYPE

// ---- 01_Equipement_Library/Operation Meter/PM_PM5XXX.TcDUT
///////////
// Structure for Schneider PM models : PM5560, PM5563, PM5563RD. Main Operating Data to be saved (ex: OPC).  
//////////
TYPE PM_PM5XXX :
STRUCT
	
	MesData					: PM ; 
                        	
	MesEAppCons				: REAL; (*(kVArh) Recieved apparent energy           	*)
	MesEAppProd				: REAL; (*(kWh) Delivered apparent energy            	*)
	                    	                                                     	
	MesUnbalanced_I1		: REAL; (*(%) Unbalanced current phase 1			 	*)
	MesUnbalanced_I2		: REAL; (*(%) Unbalanced current phase 2			 	*)
	MesUnbalanced_I3		: REAL; (*(%) Unbalanced current phase 3			 	*)	
	                    	                                                     	
	MesUnbalanced_U12		: REAL; (*(%) Unbalanced voltage U12			 	 	*)
	MesUnbalanced_U23		: REAL; (*(%) Unbalanced voltage U23				 	*)
	MesUnbalanced_U31		: REAL; (*(%) Unbalanced voltage U31				 	*)	
	                    	                                                     	
	MesUnbalanced_V1		: REAL; (*(%) Unbalanced voltage phase 1			 	*)
	MesUnbalanced_V2		: REAL; (*(%) Unbalanced voltage phase 2			 	*)
	MesUnbalanced_V3		: REAL; (*(%) Unbalanced voltage phase 3			 	*)	
		                	
	MesTHD_I1 				: REAL;	(* (%) Current Total Harmonic Distortion Phase 1. THD = (RMS of harmonics / RMS of fundamental) * 100 *)
	MesTHD_I2 				: REAL;	(* (%) Current Total Harmonic Distortion Phase 2. THD = (RMS of harmonics / RMS of fundamental) * 100 *)
	MesTHD_I3 				: REAL;	(* (%) Current Total Harmonic Distortion Phase 3. THD = (RMS of harmonics / RMS of fundamental) * 100 *)
	MesTHD_In				: REAL; (* (%) Current Total Harmonic Distortion In. THD = (RMS of harmonics / RMS of fundamental) * 100 	  *)
		                	
	MesTHD_U12				: REAL;	(* (%) Voltage U12 Total Harmonic Distortion Phase 1. THD = (RMS of harmonics / RMS of fundamental) * 100 *)
	MesTHD_U23				: REAL;	(* (%) Voltage U23 Total Harmonic Distortion Phase 2. THD = (RMS of harmonics / RMS of fundamental) * 100 *)
	MesTHD_U31				: REAL;	(* (%) Voltage U31 Total Harmonic Distortion Phase 3. THD = (RMS of harmonics / RMS of fundamental) * 100 *)
	                    	
	MesTHD_V1 				: REAL;	(* (%) Voltage V1 Total Harmonic Distortion Phase 1 - Neutre *)
	MesTHD_V2 				: REAL;	(* (%) Voltage V2 Total Harmonic Distortion Phase 2 - Neutre *)
	MesTHD_V3 				: REAL;	(* (%) Voltage V3 Total Harmonic Distortion Phase 3 - Neutre *)
	
// Alarmes 	
	MesAlarmImax			: UINT;	(* (NA) Phase over current   *) 
	MesAlarmImin 			: UINT;	(* (NA) Phase under current  *) 
	MesAlarmInmax 			: UINT;	(* (NA) Neutral over current *) 
	MesAlarmIgmax			: UINT;	(* (NA) Ground over current  *) 
	MesAlarmUmax			: UINT;	(* (NA) L-L over voltage     *) 
	MesAlarmUmin			: UINT;	(* (NA) L-L under voltage    *) 
	MesAlarmVmax			: UINT;	(* (NA) L-N over voltage     *) 
	MesAlarmVmin			: UINT;	(* (NA) L-N under Voltage    *) 
	MesAlarmPmax			: UINT;	(* (NA) Over active Power    *) 
	MesAlarmQmax			: UINT;	(* (NA) Over reactive Power  *) 
	MesAlarmSmax			: UINT;	(* (NA) Over apparent Power  *) 
	MesAlarmFreqmax			: UINT;	(* (NA) Over frequency	     *) 
	MesAlarmFreqmin			: UINT;	(* (NA) Under frequency	     *)		
	MesAlarm_PhaseLoss  	: UINT; (* (NA) Phase loss			 *) 
	MesAlarm_PhaseReversal  : UINT; (* (NA) Phase reversal		 *)	
	MesAlarmReset  			: UINT; (* (NA) PM reset 			 *) 
 	
	MesAlarmSW_Open			: BOOL; (* (NA) PM switch open 	TO BE CLARIFIED	 *)		
									 
END_STRUCT
END_TYPE

// ---- 01_Equipement_Library/Operation Meter/PM_Prometer.TcDUT
TYPE PM_Prometer :
STRUCT
		//MesData 					: PM;
	

	    F11 	: PM;       // F11                                           								
       	F15 	: PM;           // F15                                             								                               								
       	F21 	: PM;                                                 								
       	F22 	: PM;   
       	T1 	: PM;                                                 								
       	T2 	: PM;                                                 								
       	T4	: PM;
		T5 	: PM;    
	
	
	
END_STRUCT
END_TYPE

// ---- 01_Equipement_Library/Operation Meter/PM_Standard.TcDUT
///////////
// Structure For I35. Main Operating Data to be saved (ex: OPC).  
//////////
TYPE PM_Standard :
STRUCT
		MesData						: PM ; (* Object *) 
	
END_STRUCT
END_TYPE

// ---- 01_Equipement_Library/Operation Meter/PM_PM800.TcDUT
TYPE PM_PM800 :
STRUCT
	MesData 					: PM;
	
	MesTHD1 			: REAL;	(* Total Harmonic Distortion Phase 1, Adr 1199 *)
	MesTHD2 			: REAL;	(* Total Harmonic Distortion Phase 2, Adr 1200 *)
	MesTHD3 			: REAL;	(* Total Harmonic Distortion Phase 3, Adr 1201 *)
	MesTHD1N 			: REAL;	(* Total Harmonic Distortion Phase 1 - Neutre, Adr 1206 *)
	MesTHD2N 			: REAL;	(* Total Harmonic Distortion Phase 2 - Neutre, Adr 1207 *)
	MesTHD3N 			: REAL;	(* Total Harmonic Distortion Phase 3 - Neutre, Adr 1208 *)
END_STRUCT
END_TYPE

// ---- 01_Equipement_Library/Datalogger/Datalogger_PPCVerrerie.TcDUT
TYPE Datalogger_PPCVerrerie :
STRUCT
	MesData			: Datalogger ; 

	
	//225 kV 
//	PM_225kV									: PM ; // ION non remonté 
                                    			
	ProtectRelay_MainHVCB						: ProtectRelay_S42 ; 
	MainHVCB									: CB_MainHVCB_Sch ; 
                                    			
//	A1_GridHVCB									: GridHVCB ; Non remonté ? 
                                    			
	ProtectRelay_Transfo225kV					: ProtectRelay_T87 ; 
	Transfo_225kV								: Transfo_HV ; 	
	GRID										: GRID ; // non remonté ? 
	                                			
	                                			
                                    			
//	20 kV 		                    			
	MainMVCB									: CB_MainMVCB_Sch ; 
	ProtectRelay_MainMVCB						: ProtectRelay_S42 ; 
						            			
	ProtectRelay_FeederMVCB						: ARRAY[1..2] OF ProtectRelay_S42 ; 		// 1. Midi 2. Plat 
	FeederMVCB									: ARRAY[1..2] OF CB_FeederMVCB_Sch ; 
	                                	
                                    	
	                                	
	// Aux                          	
	Transfo_Aux									:  Transfo_MV ; 
	                                			
	UPS_CE										: UPS_VERR ; 
	UPS_TCM										: UPS_VERR ; 
	TapChanger 									: TapChanger ; 
	FSS											: FSS; 				(*Fire System*)
	DS											: TOR ; 			(*Door Sensor*)
	ES											: TOR ; 			(*Emergency Stop*)
	

	// Substation
	MesState									: WORD ; 			// Calculated  State of the HV + MV substation. 


	                                    		                   
	// 20 kV Courant Neutre et Cuve                                
    // transfo          ?????                                                    
	Mes20kVCourNeutCuveDefaultMasseCuve1		: BOOL;            	(*CourNeutCuveDefaultMasseCuve1	 	 *)
	Mes20kVCourNeutCuveMaxIexp2					: BOOL;            	(*CourNeutCuveMaxIexp2				 *)
	Mes20kVCourNeutCuveDefaultMasseCuve2		: BOOL;            	(*CourNeutCuveDefaultMasseCuve2	 	 *)
	Mes20kVCourNeutCuveMaxIexp4					: BOOL;            	(*CourNeutCuveMaxIexp4				 *)
	Mes20kVCourNeutCuveDefaultGround			: BOOL;            	(*CourNeutCuveDefaultGround		 	 *)
	Mes20kVCourNeutCuveMaxI0exp4				: BOOL;            	(*CourNeutCuveMaxI0exp4			 	 *)
	Mes20kVCourNeutCuveTempAlarm				: BOOL;            	(*CourNeutCuveTempAlarm			 	 *)
	Mes20kVCourNeutCuveTempTrigger				: BOOL;            	(*CourNeutCuveTempTrigger			 *)
	Mes20kVCourNeutCuveGazDischarge				: BOOL;            	(*CourNeutCuveGazDischarge			 *)
	Mes20kVCourNeutCuvePressure					: BOOL;   		   	(*CourNeutCuvePressure				 *)
	                                    		                   	
	Mes20kVCourNeutCuveI1						: REAL;            	(*(A) CourNeutCuveI1			 *)
	Mes20kVCourNeutCuveResidualI				: REAL;            	(*(A) CourNeutCuveResidualI	     *)
	Mes20kVCourNeutCuveDecltI1					: REAL;            	(*(A) CourNeutCuveDecltI1		 *)
	Mes20kVCourNeutCuveDecltI2					: REAL;            	(*(A) CourNeutCuveDecltI2		 *)
	                                                               	
	// Aux HT, BT and Transfo                                      	
	 // AuxMVCB                                                    	          
	MesAuxHTSect225kV							: BOOL;		       	(* AuxHTSect225kV						*)
	MesAuxHtSmaltHTBOpen						: BOOL;		       	(* AuxHtSmaltHTBOpen					*)
	MesAuxHtFusionFuseMeasures225kV				: BOOL;		       	(* AuxHtFusionFuseMeasures225kV			*)                                              
	MesAuxHtFusionFuseProtect225kV				: BOOL;		       	(* AuxHtFusionFuseProtect225kV			*)
	MesAuxHtFusionFuseCountRte225kV				: BOOL;		       	(* AuxHtFusionFuseCountRte225kV			*)
	MesAuxHtShortCircuitCurrentProtectCcp2		: BOOL;		       	(* AuxHtShortCircuitCurrentProtectCcp2	*)
	MesAuxHtDisjCount20kVOpen					: BOOL;		       	(* AuxHtDisjCount20kVOpen				*)
	MesAuxHtDisjRefVoltage20kVOpen				: BOOL;		       	(* AuxHtDisjRefVoltage20kVOpen			*)
	MesAuxHtShortCircuitCurrentProtectCcp3		: BOOL;		       	(* AuxHtShortCircuitCurrentProtectCcp3	*)
                                                                   	
	MesAuxBtTriggerGeneralDisj					: BOOL;		       	(*AuxBtTriggerGeneralDisj				 *)
	MesAuxBt400VManqueAC						: BOOL;		       	(*AuxBt400VManqueAC					     *)
	MesAuxBt400VDecltAntenneScada				: BOOL;		       	(*AuxBt400VDecltAntenneScada			 *)
	MesAuxBt400VDecltAntennePrio				: BOOL;		       	(*AuxBt400VDecltAntennePrio			 	 *)
	MesAuxBt400VPermutAutoStopMode				: BOOL;		       	(*AuxBt400VPermutAutoStopMode			 *)
	MesAuxBt400VPermutAutoNormalMode			: BOOL;		       	(*AuxBt400VPermutAutoNormalMode		 	 *)
	MesAuxBt400VPermutAutoSecoursMode			: BOOL;		       	(*AuxBt400VPermutAutoSecoursMode		 *)
	MesAuxBt400VPermutModeAuto					: BOOL;    	       	(*AuxBt400VPermutModeAuto				 *)
	MesAuxBt400VVoltageLossNormalAlim			: BOOL;		       	(*AuxBt400VVoltageLossNormalAlim		 *)
	MesAuxBt400VVoltageLossSecoursAlim			: BOOL;		       	(*AuxBt400VVoltageLossSecoursAlim		 *)
	MesAuxBt400VDefaultPermut					: BOOL;		       	(*AuxBt400VDefaultPermut				 *)


	MesAuxBtDefaultInverter						: BOOL;  		   	(* AuxBtDefaultInverter	*)
                                                                   	
	MesAuxBtSyntDefaultDistrib48VccJdb			: BOOL;  		   	(* AuxBtSyntDefaultDistrib48VccJdb		*)
	MesAuxBtSyntOpenDistrib48VccJdb				: BOOL;		       	(* AuxBtSyntOpenDistrib48VccJdb			*)
	MesAuxBtSyntDefaultDistrib48VccLocker		: BOOL;  		   	(* AuxBtSyntDefaultDistrib48VccLocker	*)
    MesAuxBtSyntOpenDistrib48VccLocker			: BOOL;		       	(* AuxBtSyntOpenDistrib48VccLocker		*)
                                                                   	
	MesAuxTransfoMeltingFusesContact			: BOOL;		       	(* AuxTransfoMeltingFusesContact	*)
                                                                   	
	MesAuxTransfoSwitchGear						: BOOL;	           	(*AuxTransfoSwitchGear		 *)
                                                                   	
	MesAuxHtOpenSectLine225kV					: BOOL;		       	(* AuxHtOpenSectLine225kV*)
	MesAuxHtCloseSectLine225kV					: BOOL;		       	(* AuxHtCloseSectLine225kV*)
                                                                   	
	                                                               	
	MesAuxHtOpenSectMalt						: BOOL;		       	(* AuxHtOpenSectMalt*)
	MesAuxHtCloseSectMalt						: BOOL;		       	(* AuxHtCloseSectMalt*)
                                                                   	
	MesAuxHtTeleCondamnSl225kV				 	: BOOL;		       	(* AuxHtTeleCondamnSl225kV			*)
	MesAuxHtDeTeleCondamnSl225kV				: BOOL;            	(* AuxHtDeTeleCondamnSl225kV		*)
	MesAuxHtTelecommandeRelestActif				: BOOL;		       	(* AuxHtTelecommandeRelestActif		*)
	MesAuxHtTelecommandeRelestPassif			: BOOL;	           	(* AuxHtTelecommandeRelestPassif	*)
	                                                               
	// Door Sensor, Fire Alarm, Local/Remote, Emergency Stop	   
	                                                            
	MesLocalRemoteOperation                  	: BOOL;            	(*LocalRemoteOperation    *)


	MesAlarmCom									: BOOL ; 		   	(* Communication Error with I35 module *) 

	MesAlarmCode1								: WORD ; 			(* Internal Akuo Alarm Code   *)
	MesAlarmCode2								: WORD ; 			(* Internal Akuo Alarm Code   *)
	MesAlarmCode3								: WORD ; 			(* Internal Akuo Alarm Code   *)
	MesWarningCode1								: WORD ; 			(* Internal Akuo Warning Code *)
	MesWarningCode2								: WORD ; 			(* Internal Akuo Warning Code *)  
	MesWarningCode3								: WORD ; 			(* Internal Akuo Warning Code *)
	MesWarningCode4								: WORD ; 			(* Internal Akuo Warning Code *)  
	MesWarningCode5								: WORD ; 			(* Internal Akuo Warning Code *) 
    MesWarningCode6								: WORD ; 			(* Internal Akuo Warning Code *)     
	MesEventCode1								: WORD ; 			(* Internal Akuo Event Code   *)  
	MesEventCode2								: WORD ; 			(* Internal Akuo Event Code   *) 
	MesEventCode3								: WORD ; 			(* Internal Akuo Event Code   *)  			                                                   			                                               
	
END_STRUCT
END_TYPE

// ---- 01_Equipement_Library/Operation Meter/PM_Q100.TcDUT
TYPE PM_Q100 :
STRUCT
	//Device Status 
	MesState1		: WORD ;	(* Bit0: 1=Decide OK, Bit2: 0=Battery OK, Bit4:	1=SD card error, Bit8: 1= Parameter load is in progress, Bit10: 1=	parameter check is in progress, Bit12: 1=Parameter ativation is in progress *)
	MesState2		: WORD;		(* Bit0:	1= rotation is clockwis	*)
	                            
	MesData			: PM;       (**)
                                
	MesVN			: REAL;		(*  (V) Voltage neutral conductor  *)
	CalTanPhi		: REAL;		(*  (NA) TanPhi                    *)
	MesCosPhiA		: REAL;		(*  (NA) Active power factor a     *)
	MesCosPhiB		: REAL;		(*  (NA) Active power factor b     *)
	MesCosPhiC		: REAL;		(*  (NA) Active power factor c     *)
	MesCosPhi		: REAL;		(*  (NA) Active power factor       *)
	MesEPerPulse	: REAL;		(*  (Wh, VArh, VAh per pulse) COnversion factor of counter pulses into energy values    *)
	                            
	MesEac1_dmd		: REAL;		(* Active energy based on active power Pa Demand	Counter  *)
	MesEac2_dmd		: REAL;		(* Active energy based on active power Pb Demand	Counter  *)
	MesEac3_dmd		: REAL;		(* Active energy based on active power Pc Demand Counter     *)
	MesEac_dmd		: REAL;		(* Active energy based on active power Pa Demand Counter     *)
								                                                             
	MesEac1_sup		: REAL;		(* Active energy based on active power Pa Supply Counter     *)
	MesEac2_sup		: REAL;		(* Active energy based on active power Pb Supply Counter     *)
	MesEac3_sup		: REAL;		(* Active energy based on active power Pc Supply Counter     *)
	MesEac_sup		: REAL;		(* Active energy based on active power P Supply Counter      *)
								                                                                   
	MesEreac1_cap	: REAL;		(* Reactive energy based on reactive power Qa capacitive Counter   *)
	MesEreac2_cap	: REAL;		(* Reactive energy based on reactive power Qb capacitive Counter   *)
	MesEreac3_cap	: REAL;		(* Reactive energy based on reactive power Qc capacitive Counter   *)
	MesEreac_cap	: REAL;		(* Reactive energy based on reactive power Q capacitive Counter    *)
								                                                                   
	MesEreac1_ind	: REAL;		(* Reactive energy based on reactive power Qa inductive Counter    *)
	MesEreac2_ind	: REAL;		(* Reactive energy based on reactive power Qb inductive Counter    *)
	MesEreac3_ind	: REAL;		(* Reactive energy based on reactive power Qc inductive Counter    *)
	MesEreac_ind	: REAL;		(* Reactive energy based on reactive power Q  inductive Counter    *)
								                                                                   
	CalEac1_dmd		: REAL;		(* Active energy based on active power Pa Demand         *)
	CalEac2_dmd		: REAL;		(* Active energy based on active power Pb Demand         *)
	CalEac3_dmd		: REAL;		(* Active energy based on active power Pc Demand         *)
	CalEac_dmd		: REAL;		(* Active energy based on active power Pa Demand         *)
								                                                         
	CalEac1_sup		: REAL;		(* Active energy based on active power Pa Supply         *)
	CalEac2_sup		: REAL;		(* Active energy based on active power Pb Supply         *)
	CalEac3_sup		: REAL;		(* Active energy based on active power Pc Supply         *)
	CalEac_sup		: REAL;		(* Active energy based on active power P Supply          *)
								                                                         
	CalEreac1_cap	: REAL;		(* Reactive energy based on reactive power Qa capacitive *)
	CalEreac2_cap	: REAL;		(* Reactive energy based on reactive power Qb capacitive *)
	CalEreac3_cap	: REAL;	    (* Reactive energy based on reactive power Qc capacitive *)
	CalEreac_cap	: REAL;	    (* Reactive energy based on reactive power Q capacitive  *)
								                                                         
	CalEreac1_ind	: REAL;	    (* Reactive energy based on reactive power Qa inductive  *)
	CalEreac2_ind	: REAL;	    (* Reactive energy based on reactive power Qb inductive  *)
	CalEreac3_ind	: REAL;	    (* Reactive energy based on reactive power Qc inductive  *)
	CalEreac_ind	: REAL;	    (* Reactive energy based on reactive power Q  inductive  *)
		
	MesAlarmCodeAkuo			: WORD;		(* Akuo Custom AlarmCode	*)
	MesWarningCodeAkuo			: WORD;		(* Akuo Custom WarningCode	*)
	
	

END_STRUCT
END_TYPE

// ---- 01_Equipement_Library/PCS/DCInputs_PE.TcDUT
///////////
// Structure For PE Disconecting Unit 
//////////
TYPE DCInputs_PE :
STRUCT
		
	MesIdc				: REAL ; (* (A) DC Current SV10.2   *)
//	MesUdc				: REAL ; // (V) DC Voltage 	
//	MesIDState			: WORD ; // (NA) DU State
	
END_STRUCT
END_TYPE

// ---- 01_Equipement_Library/PCS/PCS.TcDUT
///////////
// Structure for CtrlPcs Jema .  
//////////
TYPE PCS :
STRUCT

// PCS Controller  Measures



	MesState_Precharge			: BOOL;			(* (NA) Precharge indicator   - True = precharge in progress  *)
	MesOpened_Dc				: BOOL;			(* (NA) Dc Breaker status     *)
    MesOpened_Ac				: BOOL; 		(* (NA) Ac Breaker status*)

	MesAlarmCom					: BOOL; 		(* (NA) PCS Controller Communication fault*)
	MesWarningCom				: BOOL;			(* (NA) PCS Controller Communication warning*)


	
// PCS Controller  Measures
	MesP 						: REAL;  		(* (kW)  Active Power *)
	MesQ 						: REAL;  		(* (kVAr) Reactive Power*)
	MesS 						: REAL;  		(* (kVA)  Apparent Power *)
	MesPdc 						: REAL;  		(* (kW)  DC Power *)
	MesCosPhi 					: REAL;  		(* (p.u) Power factor*)
	MesU 						: REAL;  		(* (V) 	AC Voltage measure*)
	MesFreq						: REAL;			(* (Hz) Main Bus Freq*)
	MesUdc 						: REAL;  		(* (V) 	DC Voltage measure*)
	MesI 						: REAL; 		(* (A) 	Total AC current *)
	MesIdc 						: REAL; 		(* (A) 	Total DC current from batteries (+ = discharge)*)
	MesState					: WORD;			(* (NA) [P,H,B] Bit0: 1 = Not Available (AC or DC breaker open or AllAcContactorsOpened), Bit1: GridMode: 1=grid*)
	MesTemp						: REAL;			(* (°C) Temperature sensor. INV: SV4.1.4 *)


	MesSmax_ChargeFromBat		: REAL;			(* (kVA) Max apparent power available for Charge based on load factor*)
	MesSmax_DischargeFromBat	: REAL;			(* (kVA) Max apparent power available for discharge based on load factor*)

	MesPmax_ChargeFromBat		: REAL;
	
	MesPmax_DischargeFromBat	: REAL;
	
	MesID_State_Inv				: UINT;			(* (NA) Operation flag from PCS*)

	MesNbPowerColConnected		: UINT; 		(* (NA) Number of online Power Columns . SV9.1.2*)
	MesALOPowerCol_Connected	: BOOL; 		(* (NA) At least one Power Column is connected and not in alarm*)

	MesAlarm					: BOOL ; 		(* (NA) PCS Controller general Alarm*)
	MesWarning 					: BOOL; 		(* (NA) PCS Controller general Warning *)

	MesOnGrid 					: BOOL; 		(* (NA) TRUE if AFE in ONgrid Mode.*)
	MesOffGrid 					: BOOL; 		(* (NA) TRUE if AFE in Offgrid Mode.                 	*)
	MesFreqReg_Active			: BOOL; 		(* (NA) Is the frequency regulation active : True = FreqReg Active*)
	MesUReg_Active				: BOOL; 		(* (NA) Is the voltage regulation active : True = UReg Active*)
	MesSnom						: REAL; 		(* (kW) Nominal power read on Controller*)
	MesAvailability				: REAL; 		(* (%) Availability of the inverter*)

	MesAlarmCode				: WORD;			(* (NA) Internal Akuo AlarmCode*)
	MesWarningCode				: WORD; 		(* (NA) Internal Akuo WarningCode*)
	MesEventCode				: WORD;			(* (NA) Internal Akuo EventCode*)
	MesID_OpSttAlarm					: WORD ; (* SMA Operation State ENUM *)
	MesID_OpStt1Alarm				: WORD ; (* SMA Operation State 2  ENUM *)
	MesID_DrtSttAlarm				: WORD ; (* SMA Power Derating  ENUM *)
	MesID_PwrOffReas1Alarm			: WORD ; (* SMA Power Off Reason 1 ENUM *)
	MesID_PwrOffReas2Alarm 			: WORD ; (* SMA Power Off Reason 2 ENUM *)	
	
	OUT_CmdStop					: BOOL; 		(* (NA) Stop  sent to the Controller*)
	OUT_CmdStart				: BOOL;			(* (NA) Start sent to the Controller*)
	OUT_CmdStandby				: BOOL;			(* (NA) Soft stop sent to the Controller*)
	OUT_CmdPcsLocal				: BOOL;			(* (NA) If true, INV is excluded from regulation*)

	OUT_SetptP					: REAL; 		(* (kW) Active power setpoint *)

	OUT_SetptSMax				: REAL;			(* (kVA) Maximum Apparent Power setpoint*)
	OUT_SetptPMax				: REAL;			(* (kW) Upper range of the Active Power setpoint*)
	OUT_SetptPMin				: REAL;			(* (kW) Lower range of the Active Power setpoint*)

